# B&R Automation Studio project PLC code - cp (part 5)

#### MachineState.st
```iecst
ACTION MachineState:

	//Alignment photocells process
	tonAlignmentProcess.IN := (data.status.iSystemState=STP_CHECK_ALIGNMENT_STEP_3);
	tonAlignmentProcess.PT := t#2S;
	tonAlignmentProcess();

	CASE data.status.iSystemState OF

		STP_NOT_INITIALIZED:
			ResetCommands;
			ResetPhotocellAlignment;
			data.status.xReferencing :=	FALSE;

			IF NOT data.status.xReferenced THEN
				data.status.xSensorValidAlignPos := data.parameters.AlignmentProcess = STP_ALIGNMENT_NO_REQUIRED;
			END_IF

			RemoveOrderMoveAbsolute;
			SetStopOrder;
			IF xMotorStopped THEN
				RemoveStopOrder;
				CheckControllerReady;
				IF xControllerReady THEN
					data.status.iSystemState:=STP_POWER_ON;
				END_IF
			END_IF

		STP_POWER_ON:
			SetPowerOn;
			// It does HomeDirect to steppers when are power up is done
			CheckPowerOn;
			CASE data.parameters.MotorType OF
				STP_STEPPER:
					IF xPoweredOn AND NOT data.status.xReferenced THEN
						// Home Direct to enable movements
						data.status.iSystemState:=STP_HOME_DIR;

						// When Phocells are referenced and return from Zero (Man or Auto)
					ELSIF Stepper.Status.PowerOn AND StepperGear.Status.PowerOn AND data.status.xReferenced AND StepperGear.Status.PLCopenState.StandStill THEN
						data.status.iSystemState:=STP_GEARING;
					END_IF
				STP_ICLA:
					IF xPoweredOn THEN
						//Go directly to wait homing process
						data.status.iSystemState:=STP_GEARED;
					END_IF
			END_CASE

		STP_HOME_DIR:
			// Home position. Just send the order when the axis is ready
			IF Stepper.Status.PLCopenState.StandStill THEN
				Stepper.Parameter.HomePosition:=30;
				Stepper.Command.HomeDirect:=TRUE;
			END_IF
			IF StepperGear.Status.PLCopenState.StandStill THEN
				StepperGear.Parameter.HomePosition:=30;
				StepperGear.Command.HomeDirect:=TRUE;
			END_IF

			IF Stepper.Status.HomeOK AND StepperGear.Status.HomeOK THEN
				data.status.iSystemState:=STP_GEARING;
			END_IF

		STP_GEARING:
			StepperGear.Parameter.GearRatioNum:=1;
			StepperGear.Parameter.GearRationDen:=1;

			IF StepperGear.Status.PLCopenState.StandStill THEN
				StepperGear.Command.Move.GearIn:=TRUE;
			ELSIF StepperGear.Status.PLCopenState.SynchronizedMotion THEN
				data.status.iSystemState:=STP_GEARED;
			END_IF

		STP_GEARED:
			IF EDGEPOS(data.commandsSw.xReference) AND data.status.xAllPhotoInactive THEN
				data.commandsSw.xReference := FALSE;
				data.status.iSystemState := STP_HOMING_STEP_1;
			END_IF

			CheckMotorReady;
			IF data.status.xReferenced AND xMotorReady THEN
				CASE data.parameters.AlignmentProcess OF
					STP_ALIGNMENT_NO_REQUIRED:
						data.status.iSystemState := STP_STANDSTILL;

					STP_ALIGNMENT_REQUIRED:
						IF data.status.xSensorValidAlignPos THEN
							data.status.iSystemState := STP_STANDSTILL;
						ELSIF data.status.xReferencing THEN
							data.status.iSystemState := STP_SEARCH_ALIGNMENT_POS_STEP_1;
						END_IF
				END_CASE
			END_IF

			IF xMotorReady AND data.commands.Mode.xManual AND
				(data.ordersSw.xMoveDown OR data.ordersSw.xMoveUp) THEN
				data.status.iSystemState:=STP_JOGGING;
			END_IF

		STP_HOMING_STEP_1:
			data.status.xReferencing := TRUE;
			data.status.xReferenced	:= FALSE;

			IF data.parameters.xHomingEnabled THEN

				SetOrderGoingDown;

				//Stop going down when sensor to reference detects
				IF data.Inputs.Signals.xPhotoCells[data.parameters.iSensorToReference] THEN
					RemoveOrderGoingDown; // Launched stop movement

					//Once the jog is finished, we need to move up slowly to get the real position
					CheckMotorReady;
					IF xMotorReady THEN
						data.status.iSystemState := STP_HOMING_STEP_2;
					END_IF
				END_IF
			END_IF

		STP_HOMING_STEP_2:
			SetOrderGoingUp; // Launched movement

			//Moving slowly up to get the sensor again
			IF NOT data.Inputs.Signals.xPhotoCells[data.parameters.iSensorToReference] THEN
				// Movements finished
				RemoveOrderGoingUp; // Launched stop movement
				data.Alarms.xIncoherPhotocellSystem := FALSE;

				//Once the jog is finished, we need to gearOut to be able to do the Homing
				CheckMotorReady;
				IF xMotorReady THEN

					CASE data.parameters.MotorType OF
						STP_STEPPER:
							//Calculate the pulses of the HomingPosition
							MotorDriveUnit.HomePositionDesired:=data.parSw.rThicknessReference;
							MotorDriveUnit.Calculation:=CALC_HOMEPOS_PULSES;
							MotorDriveUnit();

							Stepper.Parameter.HomePosition := MotorDriveUnit.pulsesHomePositionDesired;
							StepperGear.Parameter.HomePosition := Stepper.Parameter.HomePosition;
							StepperGear.Command.Move.GearOut := TRUE;
							data.status.iSystemState := STP_HOMING_STEP_3;

						STP_ICLA:
							//Calculate the pulses of the HomingPosition
							MotorDriveUnit.HomePositionDesired:=(-1) * data.parSw.rThicknessReference;
							MotorDriveUnit.Calculation:=CALC_HOMEPOS_PULSES;
							MotorDriveUnit();

							IF Icla.Status.iActualVelocity = 0 THEN
								Icla.Parameter.Home.Position := REAL_TO_DINT(MotorDriveUnit.pulsesHomePositionDesired);
								Icla.Command.Home := TRUE;
							END_IF

							IF Icla.Status.xReferenced THEN data.status.iSystemState := STP_HOMING_STEP_3; END_IF

					END_CASE
				END_IF
			END_IF

		STP_HOMING_STEP_3:
			CASE data.parameters.MotorType OF
				STP_STEPPER:
					//Send a QuickStop to avoid the ContinuousMotion status after the GearOut
					StepperGear.Command.QuickStop := StepperGear.Status.PLCopenState.ContinuousMotion;

					IF Stepper.Status.PLCopenState.StandStill AND StepperGear.Status.PLCopenState.StandStill THEN
						// Home Direct
						Stepper.Command.HomeDirect:=TRUE;
						StepperGear.Command.HomeDirect:=TRUE;
						data.status.iSystemState := STP_HOMING_STEP_4;
					END_IF

				STP_ICLA:
					IF ABS(rPositionMotorMm - data.parSw.rThicknessReference) < 0.10 THEN
						//data.status.xReferencing := FALSE;
						data.status.xReferenced	:= TRUE;
						data.status.iSystemState := STP_GEARED;
					ELSE
						Icla.Command.Home := FALSE;
						data.status.iSystemState := STP_HOMING_STEP_2;
					END_IF
			END_CASE

		STP_HOMING_STEP_4:
			IF EDGEPOS(Stepper.Status.HomeOK AND StepperGear.Status.HomeOK) THEN
				data.status.xReferencing := FALSE;
				data.status.xReferenced	:= TRUE;
				data.status.iSystemState := STP_GEARING;
			END_IF

		STP_SEARCH_ALIGNMENT_POS_STEP_1:
			xAlignmentPositionSet := FALSE;
			SetOrderGoingUp;
			// Gauge is going to be higher than this position. Checking SensorToReference state from it.
			IF (rPositionMotorMm > data.parameters.rSensorPositionSearchAlignment) AND (data.Inputs.Signals.xPhotoCells[data.parameters.iSensorToReference]) THEN
				RemoveOrderGoingUp; // Launched stop movement
				data.status.iSystemState := STP_SEARCH_ALIGNMENT_POS_STEP_2;
			END_IF

		STP_SEARCH_ALIGNMENT_POS_STEP_2:
			SetOrderGoingUp; //Moving slowly up to get the sensor again
			IF NOT data.Inputs.Signals.xPhotoCells[data.parameters.iSensorToReference] THEN
				RemoveOrderGoingUp; // Launched stop movement
				rSensorPositionAlignmentMin := rPositionMotorMm;
				data.status.iSystemState := STP_SEARCH_ALIGNMENT_POS_STEP_3;
			END_IF

		STP_SEARCH_ALIGNMENT_POS_STEP_3:
			SetOrderGoingUp; //Moving slowly up to get the sensor again
			IF (data.Inputs.Signals.xPhotoCells[data.parameters.iSensorToReference]) THEN
				RemoveOrderGoingUp; // Launched stop movement
				rSensorPositionAlignmentMax := rPositionMotorMm;
				SetAlignmentPosition;
				data.status.rSensorPositionAlignment := rSensorPositionAlignment;
				data.status.xReferencing := FALSE;
				data.status.iSystemState := STP_STANDSTILL;
			END_IF

		STP_STANDSTILL:
			CheckAnyManualOrder;
			IF EDGEPOS(data.commandsSw.xReference) AND data.status.xAllPhotoInactive THEN
				data.commandsSw.xReference	:= FALSE;
				data.status.xReferenced	:= FALSE;
				data.status.xSensorValidAlignPos := FALSE;
				data.status.iSystemState	:= STP_HOMING_STEP_1;

			ELSIF data.commands.Mode.xManual AND xAnyManualOrder THEN
				data.status.iSystemState:=STP_JOGGING;

			ELSIF data.commands.Mode.xAuto THEN
				CASE data.parameters.AlignmentProcess OF
					STP_ALIGNMENT_NO_REQUIRED:
						data.status.iSystemState := STP_AUTO;

					STP_ALIGNMENT_REQUIRED:
						//First time machine goes to AUTO mode, to check alignment
						IF  data.status.xSensorValidAlignPos AND (NOT data.status.xAlignmentChecked) THEN
							data.status.iSystemState := STP_CHECK_ALIGNMENT_STEP_1;

						ELSIF data.status.xAlignmentChecked THEN
							data.status.iSystemState := STP_AUTO;
						END_IF
				END_CASE
			END_IF

		STP_JOGGING:
			// Stopping all
			IF tonMaxTimeJogging.Q THEN
				data.ordersSw.xMoveDown		:=	FALSE;
				data.ordersSw.xMoveUp		:=	FALSE;
			END_IF

			AssignJogOrders;

			CheckMotorReady;
			CheckAnyManualOrder;
			IF data.status.xReferenced AND xMotorReady AND NOT xAnyManualOrder THEN
				data.status.iSystemState	:= STP_STANDSTILL;

			ELSIF NOT data.status.xReferenced AND xMotorReady AND NOT xAnyManualOrder THEN
				data.status.iSystemState	:= STP_GEARED;

			END_IF

		STP_AUTO:
			IF NOT data.status.xInPosition THEN
				IF data.parameters.MotorType = STP_STEPPER THEN
					MotorDriveUnit.PositionDesired := rSensorPositionDesired;
				ELSE
					MotorDriveUnit.PositionDesired := (-1) * rSensorPositionDesired;
				END_IF
				MotorDriveUnit.Calculation := CALC_POS_PULSES;
				MotorDriveUnit();
				SetOrderMoveAbsolute;
				data.status.iSystemState := STP_RUNING;
			END_IF

		STP_CHECK_ALIGNMENT_STEP_1:
			//When the movement is finished
			IF data.parameters.MotorType = STP_STEPPER THEN
				MotorDriveUnit.PositionDesired := rSensorPositionAlignment;
			ELSE
				MotorDriveUnit.PositionDesired := (-1) * rSensorPositionAlignment;
			END_IF
			MotorDriveUnit.Calculation := CALC_POS_PULSES;
			MotorDriveUnit();
			SetOrderMoveAbsolute;
			data.status.iSystemState := STP_CHECK_ALIGNMENT_STEP_2;

		STP_CHECK_ALIGNMENT_STEP_2:
			//When the movement is finished
			IF (ABS(rPositionMotorMm-rSensorPositionAlignment)<0.25)  THEN
				data.status.iSystemState := STP_CHECK_ALIGNMENT_STEP_3;
			END_IF

			//Sensor alignment checking process cancelled when print order is set
			ReviewCancelCheckAlignment;

		STP_CHECK_ALIGNMENT_STEP_3:
			IF tonAlignmentProcess.Q THEN
				CheckPhotocellsAlignment;
				tonAlignmentProcess(IN := FALSE); //Clean the timer for next time in this stage

			//Due to issue DELOREAN-1129. Motor stays in this state. To exit, go to zero mode, then "xAlignmentChecked" is set to FALSE check process is executed when going to auto again.
			ELSIF data.status.xAlignmentChecked THEN
				data.status.iSystemState := STP_CHECK_ALIGNMENT_STEP_4;
			END_IF

			//Sensor alignment checking process cancelled when print order is set
			ReviewCancelCheckAlignment;

		STP_CHECK_ALIGNMENT_STEP_4:
			IF (NOT data.Alarms.xAlrCriticalPhotocellNotAligned) OR data.commands.Mode.xZero THEN
				data.status.iSystemState := STP_CHECK_ALIGNMENT_STEP_5;
			ELSIF data.commands.xErrorRst THEN
				ResetPhotocellAlignment;
				data.status.iSystemState := STP_CHECK_ALIGNMENT_STEP_3;
			END_IF

		STP_CHECK_ALIGNMENT_STEP_5:
			// Code from AUTO (previously from STP_CHECK_ALIGNMENT_STEP_4 to StandStill>>Auto
			IF NOT data.status.xInPosition THEN
				IF data.parameters.MotorType = STP_STEPPER THEN
					MotorDriveUnit.PositionDesired := rSensorPositionDesired;
				ELSE
					MotorDriveUnit.PositionDesired := (-1) * rSensorPositionDesired;
				END_IF
				MotorDriveUnit.Calculation := CALC_POS_PULSES;
				MotorDriveUnit();
				SetOrderMoveAbsolute;
				data.status.iSystemState := STP_CHECK_ALIGNMENT_STEP_6;
			END_IF

		STP_CHECK_ALIGNMENT_STEP_6:
			// Code from RUNNING. Previously from Auto>>Running
			//If the movement is finished or the desired position has changed
			tonMotorStopped(IN:=xMotorStopped, PT:=T#500ms);
			IF (data.status.xInPosition OR tonMotorStopped.Q) THEN
				RemoveOrderMoveAbsolute;
				data.status.iSystemState := STP_AUTO;
				tonMotorStopped(IN:=FALSE);
			END_IF

		STP_RUNING:
			//If the movement is finished or the desired position has changed
			tonMotorStopped(IN:=xMotorStopped, PT:=T#500ms);
			IF (data.status.xInPosition OR tonMotorStopped.Q) THEN
				RemoveOrderMoveAbsolute;
				data.status.iSystemState := STP_AUTO;
				tonMotorStopped(IN:=FALSE);
			END_IF

		STP_ERROR:
			ResetCommands;
			SetPowerOff;

			IF data.parameters.MotorType = STP_STEPPER THEN
				Stepper.Command.Reset := Stepper.Status.ControllerReady AND Stepper.Status.ErrorID<>0 AND data.commands.xErrorRst;
				Stepper.Command.ErrorAcknowledge :=	Stepper.Status.ErrorID<>0 AND data.commands.xErrorRst;

				StepperGear.Command.Reset := StepperGear.Status.ControllerReady AND StepperGear.Status.ErrorID<>0 AND data.commands.xErrorRst;
				StepperGear.Command.ErrorAcknowledge := StepperGear.Status.ErrorID<>0 AND data.commands.xErrorRst;
			END_IF

			data.status.xReferencing :=	FALSE;

			IF NOT data.status.xMotorError THEN data.status.iSystemState:=STP_NOT_INITIALIZED; END_IF;

	END_CASE

	//Sending nLaser to ERROR
	CASE data.parameters.MotorType OF
		STP_STEPPER:
			// Force state in Error/Zero state
			IF ((xAnyErrorStepper OR data.AlSummary.xAnyAlarm) AND (Stepper.Status.ErrorID<>31221)) OR tonTimeOutGearing.Q THEN
				data.status.iSystemState:=STP_ERROR;
			END_IF

		STP_ICLA:
			IF ((Icla.Status.iDriveStatus = ICLAST_ERROR) OR data.AlSummary.xAnyAlarm) THEN
				data.status.iSystemState:=STP_ERROR;
			END_IF
	END_CASE

	//In Zero mode it goes to not Init
	IF (data.commands.Mode.xZero) THEN
		data.status.iSystemState:=STP_NOT_INITIALIZED;
	END_IF;

	iReasonCheckingAlignment.0 := data.status.iSystemState = STP_CHECK_ALIGNMENT_STEP_1;
	iReasonCheckingAlignment.1 := data.status.iSystemState = STP_CHECK_ALIGNMENT_STEP_2;
	iReasonCheckingAlignment.2 := data.status.iSystemState = STP_CHECK_ALIGNMENT_STEP_3;
	iReasonCheckingAlignment.3 := data.status.iSystemState = STP_CHECK_ALIGNMENT_STEP_4;
	iReasonCheckingAlignment.4 := data.status.iSystemState = STP_CHECK_ALIGNMENT_STEP_5;
	iReasonCheckingAlignment.5 := data.status.iSystemState = STP_CHECK_ALIGNMENT_STEP_6;
	data.status.xCheckingAlignment := iReasonCheckingAlignment > 0;

	//Silvia: delay gearing motors.
	tonTimeOutGearing.IN:=data.status.iSystemState=STP_GEARING;
	tonTimeOutGearing.PT:=t#4s;
	tonTimeOutGearing();

	//Alarm excessive photecell activated
	tonMaxTimeJogging.IN:= (data.ordersSw.xMoveDown OR data.ordersSw.xMoveUp);
	tonMaxTimeJogging.PT:= T#5S;
	tonMaxTimeJogging();

	//Saving state history
	IF data.status.iSystemState<>StateHistory[0] THEN
		FOR iIndexHistory:=iHistoryLines TO 1 BY -1 DO
			StateHistory[iIndexHistory]:=StateHistory[iIndexHistory-1];
		END_FOR;
		StateHistory[0]:=data.status.iSystemState;
	END_IF

END_ACTION

ACTION ResetCommands:
	IF data.parameters.MotorType = STP_STEPPER THEN
		StepperGear.Command.Power      := FALSE;
		Stepper.Command.QuickStop	   := FALSE;
		StepperGear.Command.QuickStop  := FALSE;
		Stepper.Command.Jog.ContinuousPos	:=	FALSE;
		Stepper.Command.Jog.ContinuousNeg	:=	FALSE;
	ELSIF data.parameters.MotorType = STP_ICLA THEN
		Icla.Command.Enable := FALSE;
		Icla.Command.JogBackward := FALSE;
		Icla.Command.JogForward := FALSE;
		Icla.Command.MoveAbsolute := FALSE;
	END_IF
	data.commandsSw := ResetCommandsSw;
END_ACTION

ACTION CheckControllerReady:
	CASE data.parameters.MotorType OF
		STP_STEPPER:
			xControllerReady := Stepper.Status.ControllerReady AND StepperGear.Status.ControllerReady;
		STP_ICLA:
			xControllerReady := NOT Icla.Status.Error.Communication;
	END_CASE
END_ACTION

ACTION SetPowerOn:
	CASE data.parameters.MotorType OF
		STP_STEPPER:
			Stepper.Command.Power:=TRUE;
			StepperGear.Command.Power:=TRUE;
		STP_ICLA:
			Icla.Command.Enable := TRUE;
	END_CASE
END_ACTION

ACTION SetPowerOff:
	CASE data.parameters.MotorType OF
		STP_STEPPER:
			Stepper.Command.Power:=FALSE;
			StepperGear.Command.Power:=FALSE;
		STP_ICLA:
			Icla.Command.Enable := FALSE;
	END_CASE
END_ACTION

ACTION CheckPowerOn:
	CASE data.parameters.MotorType OF
		STP_STEPPER:
			xPoweredOn := Stepper.Status.PowerOn AND StepperGear.Status.PowerOn;
		STP_ICLA:
			xPoweredOn := Icla.Status.IclaStatus = AXISILE_POWER OR Icla.Status.IclaStatus = AXISILE_READY;
	END_CASE
END_ACTION

ACTION CheckMotorReady:
	CASE data.parameters.MotorType OF
		STP_STEPPER:
			xMotorReady := Stepper.Status.PLCopenState.StandStill AND StepperGear.Status.PLCopenState.SynchronizedMotion;
		STP_ICLA:
			xMotorReady := Icla.Status.iDriveStatus = ICLAST_ENABLE_OPERATION;
	END_CASE
END_ACTION

ACTION SetOrderGoingDown:
	CASE data.parameters.MotorType OF
		STP_STEPPER:
			Stepper.Command.Jog.ContinuousNeg := TRUE;

		STP_ICLA:
			Icla.Command.JogForward := TRUE;
	END_CASE
END_ACTION

ACTION RemoveOrderGoingDown:
	CASE data.parameters.MotorType OF
		STP_STEPPER:
			Stepper.Command.Jog.ContinuousNeg := FALSE;

		STP_ICLA:
			Icla.Command.JogForward := FALSE;
	END_CASE
END_ACTION

ACTION SetOrderGoingUp:
	CASE data.parameters.MotorType OF
		STP_STEPPER:
			Stepper.Command.Jog.ContinuousPos := TRUE;

		STP_ICLA:
			Icla.Command.JogBackward := TRUE;
	END_CASE
END_ACTION

ACTION RemoveOrderGoingUp:
	CASE data.parameters.MotorType OF
		STP_STEPPER:
			Stepper.Command.Jog.ContinuousPos := FALSE;

		STP_ICLA:
			Icla.Command.JogBackward := FALSE;
	END_CASE
END_ACTION

ACTION SetOrderMoveAbsolute:
	CASE data.parameters.MotorType OF
		STP_STEPPER:
			Stepper.Parameter.Position := MotorDriveUnit.pulsesPositionDesired;
			Stepper.Command.Move.Absolute := TRUE;

		STP_ICLA:
			Icla.Parameter.MoveAbsolute.Position := REAL_TO_DINT(MotorDriveUnit.pulsesPositionDesired);
			Icla.Command.MoveAbsolute := TRUE;
	END_CASE
END_ACTION

ACTION RemoveOrderMoveAbsolute:
	CASE data.parameters.MotorType OF
		STP_STEPPER:
			Stepper.Command.Move.Absolute := FALSE;

		STP_ICLA:
			Icla.Command.MoveAbsolute := FALSE;

	END_CASE
END_ACTION

ACTION SetStopOrder:
	CASE data.parameters.MotorType OF
		STP_STEPPER:
			Stepper.Command.QuickStop := TRUE;

		STP_ICLA:
			Icla.Command.Stop := TRUE;

	END_CASE
END_ACTION

ACTION RemoveStopOrder:
	CASE data.parameters.MotorType OF
		STP_STEPPER:
			Stepper.Command.QuickStop := FALSE;

		STP_ICLA:
			Icla.Command.Stop := FALSE;

	END_CASE
END_ACTION

ACTION AssignJogOrders:
	CASE data.parameters.MotorType OF
		STP_STEPPER:
			Stepper.Command.Jog.ContinuousPos	:=	data.ordersSw.xMoveUp;
			Stepper.Command.Jog.ContinuousNeg	:=	data.ordersSw.xMoveDown AND NOT Stepper.Command.Jog.ContinuousPos;

		STP_ICLA:
			Icla.Command.JogForward := data.ordersSw.xMoveDown AND NOT data.ordersSw.xMoveUp;
			Icla.Command.JogBackward := NOT data.ordersSw.xMoveDown AND data.ordersSw.xMoveUp;

	END_CASE
END_ACTION

ACTION CheckAnyManualOrder:
	xAnyManualOrder := data.ordersSw.xMoveUp OR data.ordersSw.xMoveDown;
END_ACTION

ACTION SetAlignmentPosition:
	rSensorPositionAlignment := (rSensorPositionAlignmentMax + rSensorPositionAlignmentMin)/2;
	data.status.xSensorValidAlignPos := (data.parameters.rSensorMechPositionAlignmentMin < rSensorPositionAlignment) AND (rSensorPositionAlignment < data.parameters.rSensorMechPositionAlignmentMax);
	xAlignmentPositionSet := rSensorPositionAlignment>0;
END_ACTION

ACTION CheckPhotocellsAlignment:
	FOR iIndexSensor:=1 TO data.parameters.iSensorQuantity DO
		data.status.xPhotoCellsNotAligned[iIndexSensor] := data.Inputs.Signals.xPhotoCells[iIndexSensor];
	END_FOR

	data.status.xAlignmentChecked := TRUE;
END_ACTION

ACTION ResetPhotocellAlignment:
	data.status.xAlignmentChecked := FALSE;
END_ACTION

ACTION CancelAlignment:
	data.status.xAlignmentChecked := TRUE;
END_ACTION

ACTION ReviewCancelCheckAlignment:
	IF (data.commands.xCancelAlignmentCheck) THEN
		CancelAlignment;
		RemoveOrderMoveAbsolute; //Allow a new edge and going to final position
		SetStopOrder;
		IF xMotorStopped THEN
			RemoveStopOrder;
			data.status.iSystemState:=STP_STANDSTILL;
		END_IF
	END_IF
END_ACTION
```

#### Motors.st
```iecst
ACTION DataToMotors:

	data.parSw.rMechOffset:=LIMIT(-1,data.parSw.rMechOffset, 1);

	IF data.parameters.MotorType = STP_STEPPER THEN
		StepperGear.Parameter.Direction	:= Stepper.Parameter.Direction; 	(* Step for a StepByStep movement *) (*Take carewith relative movements!!!!*)
	END_IF

	rJogSpeedSetPoint:=data.parameters.JogSpeed;

	//Drive Unit Data Managment
	MotorDriveUnit.TransmissionData := data.parameters.DriveUnit;

	MotorDriveUnit.SpeedDesired:=data.parameters.Speed;
	MotorDriveUnit.Calculation:=CALC_SPEED_PULSES;
	MotorDriveUnit();

	MotorDriveUnit.JogSpeedDesired:=rJogSpeedSetPoint;
	MotorDriveUnit.Calculation:=CALC_JOGSPEED_PULSES;
	MotorDriveUnit();

	MotorDriveUnit.AccelerationDesired:=data.parameters.Acceleration;
	MotorDriveUnit.Calculation:=CALC_ACC_PULSES;
	MotorDriveUnit();

	AssignDataToMotors;

END_ACTION

ACTION AssignDataToMotors:

	CASE data.parameters.MotorType OF
		STP_STEPPER:

			//Speed
			Stepper.Parameter.Speed:=MotorDriveUnit.pulsesSpeedDesired;
			StepperGear.Parameter.Speed := Stepper.Parameter.Speed;

			//Jog Speed
			Stepper.Parameter.JogSpeed:=MotorDriveUnit.pulsesJogSpeedDesired;
			StepperGear.Parameter.JogSpeed:=Stepper.Parameter.JogSpeed;

			//Acceleration
			Stepper.Parameter.Acceleration := MotorDriveUnit.pulsesAccelerationDesired;
			Stepper.Parameter.Deceleration := Stepper.Parameter.Acceleration;
			StepperGear.Parameter.Acceleration := Stepper.Parameter.Acceleration;
			StepperGear.Parameter.Deceleration := Stepper.Parameter.Deceleration;

			//Reset
			Stepper.Command.ErrorAcknowledge:= Stepper.Status.ErrorID=31221 OR (Stepper.Status.ErrorID = 29207) OR (Stepper.Status.ErrorID = 29205); // Disturbance in cables?
			StepperGear.Command.ErrorAcknowledge:= StepperGear.Status.ErrorID=31221 OR (Stepper.Status.ErrorID = 29207) OR (Stepper.Status.ErrorID = 29205);

			//Enable Permanent Encoder Data
			Stepper.Parameter.Init.xEnabledPermEncData:=TRUE;
			StepperGear.Parameter.Init.xEnabledPermEncData:=TRUE;

		STP_ICLA:

			//Enable
			Icla.Command.Enable:= Icla.Status.iDriveStatus <> ICLAST_ERROR;

			//Speed
			Icla.Parameter.MoveAbsolute.Velocity := REAL_TO_UINT(MotorDriveUnit.pulsesSpeedDesired);

			//Jog Speed
			Icla.Parameter.Jog.VeloSlow := REAL_TO_UINT(MotorDriveUnit.pulsesJogSpeedDesired);
			Icla.Command.JogFastSpeed := FALSE;

			//Acceleration
			Icla.Parameter.iAcceleration := REAL_TO_UINT(MotorDriveUnit.pulsesAccelerationDesired);

			//Reset
			Icla.Command.Reset := 	data.commands.xResetMotor OR 	(data.commands.xErrorRst AND
																	Icla.Status.IclaStatus <> AXISILE_MOVE_ABSOLUTE AND
																	Icla.Status.IclaStatus <> AXISILE_JOG AND
																	Icla.Status.IclaStatus <> AXISILE_HOMING);

			data.status.Icla.xIsMoving := Icla.Status.iActualVelocity<>0;

	END_CASE

END_ACTION

ACTION DataFromMotors:

	CASE data.parameters.MotorType OF
		STP_STEPPER:
			// All manual movements are done with Jog, Photocells.status.xReferencing is done by Jog, could be it done by trigger?
			xAnyManualMovement:= Stepper.Status.PLCopenState.ContinuousMotion OR StepperGear.Status.PLCopenState.ContinuousMotion;

			MotorDriveUnit.pulsesDevice:=Stepper.Status.ActPosition;

			//Conversions
			MotorDriveUnit.Calculation:= CALC_POS_MM;
			MotorDriveUnit();
			rPositionMotorMm := MotorDriveUnit.PositionDevice;

			data.status.rPositionMotor := rPositionMotorMm;

			// Errrors assumed ?
			xAnyErrorStepper:=	(Stepper.Status.ErrorID<>0) OR (StepperGear.Status.ErrorID<>0);
			data.status.xMotorError:= xAnyErrorStepper AND (((Stepper.Status.ErrorID<>31221)AND (Stepper.Status.ErrorID<>29207) AND (Stepper.Status.ErrorID<>29205)) OR // It avoids data.status.xZero
															((StepperGear.Status.ErrorID<>31221)AND (StepperGear.Status.ErrorID<>29207) AND (StepperGear.Status.ErrorID<>29205)));
			data.status.iErrorId:=Stepper.Status.ErrorID;
			xMotorStopped := Stepper.Status.ActVelocity = 0;

			IF (Stepper.Status.ErrorID = 29205) OR (StepperGear.Status.ErrorID = 29205) THEN
				data.status.xReferenced := FALSE;
			END_IF

		STP_ICLA:
			xAnyManualMovement:= (Icla.Status.IclaStatus = AXISILE_JOG);

			MotorDriveUnit.pulsesDevice := DINT_TO_REAL(Icla.Status.iActualPosition);
			MotorDriveUnit.PulsesSpeedDevice:=Icla.Status.iActualVelocity;

			// Conversions
			MotorDriveUnit.Calculation:= CALC_POS_MM;
			MotorDriveUnit();
			rPositionMotorMm := (-1)*MotorDriveUnit.PositionDevice;

			data.status.rPositionMotor := rPositionMotorMm;

			// Errors
			data.status.xMotorError:= Icla.Status.Error.Communication OR Icla.Status.Error.ErrorNumber<>0; // It avoids data.status.xZero
			data.status.Icla.iErrorId:= Icla.Status.Error.ErrorNumber;

			data.status.Icla.rCurrentPosition:= Icla.Status.iActualPosition;
			data.status.Icla.rCurrentVel:= Icla.Status.iActualVelocity;

			xMotorStopped := Icla.Status.iActualVelocity = 0;

	END_CASE

	//Sending upwards the information of the location of the sensors
	data.status.xInPosition := ABS(rPositionMotorMm - rSensorPositionDesired) < 0.10;
	data.status.xAboveSetPoint := rPositionMotorMm >= rSensorPositionDesired + 0.10;
	data.status.xBelowSetPoint := rPositionMotorMm <= rSensorPositionDesired - 0.10;

	//To avoid change rBarsPosition value while motor is being positioned to new position setpoint. Issue discovered while changing thickness from 2 to 10mm at 90m/min
	//Bars were going down executing little steps because "rMaxPosition" was written every scan cycle with a new value coming due to this "rPositionWithOffset"
	IF data.status.xInPosition THEN
		data.status.rPositionWithOffset := rPositionMotorMm - data.parSw.rMechOffset;
	END_IF

	MotorDriveUnit.Calculation:= CALC_SPEED_MM;
	MotorDriveUnit();

END_ACTION
```

### Program Logical/ExtPack/_Media/nSensorCtrl/nSensorCtrl_v2/nSensorCtrl_Fast (IEC)

#### nSensorCtrl_Fast.st - Init, cyclic, exit code
```iecst
PROGRAM _CYCLIC

	//Main data assignation
	data 	ACCESS ADR (gPhotoCells);

	//Not execute the code if the nSensor system is not installed
	IF NOT data.status.xInstalled THEN	RETURN;	END_IF

	//If in not Simulation check the pointers and assign data
	IF gMachine.St.HwData.Family <> FAMILY_BRAUTOMATIONRUNTIME THEN

		// Check value for all sensors considered
		FOR iIndexCheckSensor := 1 TO data.parameters.iSensorQuantity DO
			IF (data.Inputs.Signals.pInput[iIndexCheckSensor] <> 0) THEN
				pointerValue ACCESS (data.Inputs.Signals.pInput[iIndexCheckSensor]);
				data.Inputs.Signals.xPhotoCells[iIndexCheckSensor] := NOT pointerValue;
			ELSE
				RETURN;
			END_IF
		END_FOR

	END_IF

	xRecordMaxPosition := data.commands.xRecordMaxPosition;
	IF xRecordMaxPosition THEN
		rMaxPosition := MAX(data.parameters.rMediaThickness, data.status.rPositionWithOffset);
		rBarPosition := rMaxPosition;
	END_IF

	IF data.status.xSensorsPositionedRelativeToBar THEN
		iFirstSensorToCheck:=data.status.iSensorToApplyOffset;
	ELSE
		iFirstSensorToCheck:=data.parameters.iSensorToReference;
	END_IF

	xMountedMediaDetected := FALSE;
	xMediaToRejectDetected := FALSE;

	// Checking Mounted data if machine is in conditions to Check
	IF data.commands.xCheckMounted THEN
		//Just above the Sensor for reference. Sensors below not used. Just to know if media inside (parameters.iSensorToReference)
		//Running photocells from the one assemblied closest to printer's entry and highest located. In case mountedTile alarm, will be active at first iterations
		FOR iIndexSensor:=iFirstSensorToCheck TO data.parameters.iSensorQuantity DO
			IF data.Inputs.Signals.xPhotoCells[iIndexSensor] THEN
				//Define the position of the bars
				IF iIndexSensor<>data.parameters.iSensorQuantity THEN
					IF data.status.xSensorsPositionedRelativeToBar THEN
						rBarPosition := data.status.rOffsetToApplyToBarsPosition + data.parameters.rOffsetRelToBar + data.parameters.Sensors[iIndexSensor+1].rDistanceRelativeToFirstSensor + data.parameters.Sensors[iIndexSensor+1].rSafetyOffset;
					ELSE
						rBarPosition := data.parameters.rMediaThickness + data.parameters.Sensors[iIndexSensor+1].rDistanceRelativeToFirstSensor + data.parameters.rOffsetPosition + data.parameters.Sensors[iIndexSensor+1].rSafetyOffset;
					END_IF
				END_IF

				// Define the States to raise Mounted Alarms
				iStatusCheckMounted.0 := data.status.iSystemState = STP_AUTO;
				iStatusCheckMounted.1 := data.status.iSystemState = STP_RUNING;

				IF iStatusCheckMounted > 0 THEN
					//Raise the Mounted alarm if sensor active and it is configured to raise mounted.
					IF data.parameters.xRaiseMountedJustBelowPrePrint THEN
						// This is the case for Cube_Alpha, where was important add more safety to do not raise the alarm in the wrong position and with nonsense
						IF data.parameters.Sensors[iIndexSensor].xMountedMedia AND data.status.rPositionMotor < data.parameters.rPrePrintPosition + 0.5 THEN
							// This alarm has to be raised here to avoid resetting it and move out the mounted media
							IF NOT data.commands.xMountedMediaInside THEN
								data.Alarms.xMountedTile:= TRUE;
							END_IF
							xMountedMediaDetected := TRUE;
							EXIT;
						END_IF
					ELSE
						// Previous behavior not tacking into account Cube machines
						IF data.parameters.Sensors[iIndexSensor].xMountedMedia THEN
							// This alarm has to be raised here to avoid resetting it and move out the mounted media
							IF NOT data.commands.xMountedMediaInside THEN
								data.Alarms.xMountedTile:= TRUE;
							END_IF
							xMountedMediaDetected := TRUE;
							EXIT;
						END_IF
					END_IF
				END_IF

				//Marking media to be rejected when any laser configured to do that. Due to low quality printing when bars moving up upper of sensor's height
				IF data.parSw.Sensors[iIndexSensor].xToRejectMedia THEN
					xMediaToRejectDetected := TRUE;
				END_IF

			END_IF

		END_FOR

	ELSE
		//data.status.xMediaToRejectDetected := FALSE;
	END_IF

	// Data has to be treated in the slow program to be sure to read the information in all fast programs
	IF xMountedMediaDetected (*AND NOT data._Internal.xMountedMediaTreated*) THEN
		data.status.xMountedMediaDetected := TRUE;
	ELSIF NOT xMountedMediaDetected AND data._Internal.xMountedMediaTreated THEN
		data.status.xMountedMediaDetected := FALSE;
	END_IF

	// Data has to be treated in the slow program to be sure to read the information in all fast programs
	IF xMediaToRejectDetected (*AND NOT data._Internal.xMediaToRejectTreated*) THEN
		data.status.xMediaToRejectDetected := TRUE;
	ELSIF NOT xMediaToRejectDetected AND data._Internal.xMediaToRejectTreated THEN
		data.status.xMediaToRejectDetected := FALSE;
	END_IF

	data.status.rBarsPosition := rBarPosition;
	data.status.xLowPieceDetect := data.Inputs.Signals.xPhotoCells[1];

	// If the bars are in high position, do not register photocelles activation/deactivation
	IF data.status.rPositionMotor > (data.parameters.rPrePrintPosition + 0.5) THEN
		RETURN;
	END_IF

	IF EDGEPOS(data.Inputs.Signals.xPhotoCells[2]) THEN LogRaiseSensor2; END_IF
	IF EDGEPOS(data.Inputs.Signals.xPhotoCells[3]) THEN LogRaiseSensor3; END_IF
	IF EDGEPOS(data.Inputs.Signals.xPhotoCells[4]) THEN LogRaiseSensor4; END_IF
	IF EDGEPOS(data.Inputs.Signals.xPhotoCells[5]) THEN LogRaiseSensor5; END_IF
	IF EDGEPOS(data.Inputs.Signals.xPhotoCells[6]) THEN LogRaiseSensor6; END_IF

	IF EDGENEG(data.Inputs.Signals.xPhotoCells[2]) THEN LogLowerSensor2; END_IF
	IF EDGENEG(data.Inputs.Signals.xPhotoCells[3]) THEN LogLowerSensor3; END_IF
	IF EDGENEG(data.Inputs.Signals.xPhotoCells[4]) THEN LogLowerSensor4; END_IF
	IF EDGENEG(data.Inputs.Signals.xPhotoCells[5]) THEN LogLowerSensor5; END_IF
	IF EDGENEG(data.Inputs.Signals.xPhotoCells[6]) THEN LogLowerSensor6; END_IF

END_PROGRAM
```

#### EventLog.st
```iecst
ACTION LogRaiseSensor2:

	stRaiseSensor2.Source := ELOG_TYPE_DETECTION;
	stRaiseSensor2.Severity:= ELOG_SEVERITY_INFO;
	stRaiseSensor2.Facility:= 2;
	stRaiseSensor2.ErrorCode:=0;

	stRaiseSensor2.Text := 'nSensor. Raised Sensor2';

	gEventLogLoader(EventData := ADR(stRaiseSensor2));

END_ACTION

ACTION LogLowerSensor2:

	stLowerSensor2.Source := ELOG_TYPE_DETECTION;
	stLowerSensor2.Severity:= ELOG_SEVERITY_INFO;
	stLowerSensor2.Facility:= 2;
	stLowerSensor2.ErrorCode:=0;

	stLowerSensor2.Text := 'nSensor. Lowered Sensor2';

	gEventLogLoader(EventData := ADR(stLowerSensor2));

END_ACTION

ACTION LogRaiseSensor3:

	stRaiseSensor3.Source := ELOG_TYPE_DETECTION;
	stRaiseSensor3.Severity:= ELOG_SEVERITY_INFO;
	stRaiseSensor3.Facility:= 3;
	stRaiseSensor3.ErrorCode:=0;

	stRaiseSensor3.Text := 'nSensor. Raised Sensor3';

	gEventLogLoader(EventData := ADR(stRaiseSensor3));

END_ACTION

ACTION LogLowerSensor3:

	stLowerSensor3.Source := ELOG_TYPE_DETECTION;
	stLowerSensor3.Severity:= ELOG_SEVERITY_INFO;
	stLowerSensor3.Facility:= 3;
	stLowerSensor3.ErrorCode:=0;

	stLowerSensor3.Text := 'nSensor. Lowered Sensor3';

	gEventLogLoader(EventData := ADR(stLowerSensor3));

END_ACTION

ACTION LogRaiseSensor4:

	stRaiseSensor4.Source := ELOG_TYPE_DETECTION;
	stRaiseSensor4.Severity:= ELOG_SEVERITY_INFO;
	stRaiseSensor4.Facility:= 4;
	stRaiseSensor4.ErrorCode:=0;

	stRaiseSensor4.Text := 'nSensor. Raised Sensor4';

	gEventLogLoader(EventData := ADR(stRaiseSensor4));

END_ACTION

ACTION LogLowerSensor4:

	stLowerSensor4.Source := ELOG_TYPE_DETECTION;
	stLowerSensor4.Severity:= ELOG_SEVERITY_INFO;
	stLowerSensor4.Facility:= 4;
	stLowerSensor4.ErrorCode:=0;

	stLowerSensor4.Text := 'nSensor. Lowered Sensor4';

	gEventLogLoader(EventData := ADR(stLowerSensor4));

END_ACTION

ACTION LogRaiseSensor5:

	stRaiseSensor5.Source := ELOG_TYPE_DETECTION;
	stRaiseSensor5.Severity:= ELOG_SEVERITY_INFO;
	stRaiseSensor5.Facility:= 5;
	stRaiseSensor5.ErrorCode:=0;

	stRaiseSensor5.Text := 'nSensor. Raised Sensor5';

	gEventLogLoader(EventData := ADR(stRaiseSensor5));

END_ACTION

ACTION LogLowerSensor5:

	stLowerSensor5.Source := ELOG_TYPE_DETECTION;
	stLowerSensor5.Severity:= ELOG_SEVERITY_INFO;
	stLowerSensor5.Facility:= 5;
	stLowerSensor5.ErrorCode:=0;

	stLowerSensor5.Text := 'nSensor. Lowered Sensor5';

	gEventLogLoader(EventData := ADR(stLowerSensor5));

END_ACTION

ACTION LogRaiseSensor6:

	stRaiseSensor6.Source := ELOG_TYPE_DETECTION;
	stRaiseSensor6.Severity:= ELOG_SEVERITY_INFO;
	stRaiseSensor6.Facility:= 6;
	stRaiseSensor6.ErrorCode:=0;

	stRaiseSensor6.Text := 'nSensor. Raised Sensor6';

	gEventLogLoader(EventData := ADR(stRaiseSensor6));

END_ACTION

ACTION LogLowerSensor6:

	stLowerSensor6.Source := ELOG_TYPE_DETECTION;
	stLowerSensor6.Severity:= ELOG_SEVERITY_INFO;
	stLowerSensor6.Facility:= 6;
	stLowerSensor6.ErrorCode:=0;

	stLowerSensor6.Text := 'nSensor. Lowered Sensor6';

	gEventLogLoader(EventData := ADR(stLowerSensor6));

END_ACTION
```

#### nSensorCtrl_Fast.var - Local variables
```iecst
VAR
	data : REFERENCE TO nSensors_typ;
	rMaxPosition : REAL;
	rBarPosition : REAL;
	iFirstSensorToCheck : USINT;
	iIndexSensor : USINT;
	xRecordMaxPosition : BOOL; (*Variable to allow to record the max position*)
	iStatusCheckMounted : UINT;
	xMountedMediaDetected : BOOL;
	xMediaToRejectDetected : BOOL;
	iIndexCheckSensor : USINT;
	pointerValue : REFERENCE TO BOOL;
	stRaiseSensor1 : EventLog_typ;
	stLowerSensor1 : EventLog_typ;
	stRaiseSensor2 : EventLog_typ;
	stLowerSensor2 : EventLog_typ;
	stRaiseSensor3 : EventLog_typ;
	stLowerSensor3 : EventLog_typ;
	stRaiseSensor4 : EventLog_typ;
	stLowerSensor4 : EventLog_typ;
	stRaiseSensor5 : EventLog_typ;
	stLowerSensor5 : EventLog_typ;
	stRaiseSensor6 : EventLog_typ;
	stLowerSensor6 : EventLog_typ;
	stRaiseSensor7 : EventLog_typ;
	stLowerSensor7 : EventLog_typ;

END_VAR
```

### Program Logical/ExtPack/_Media/nSensorCtrl/nSensorSim/nSensorSim_v1/nSensorSim (IEC)

#### nSensorSim.var - Local variables
```iecst
VAR
	data : REFERENCE TO nSensors_typ;
	iIndexSensor : USINT;
	rGaugeHeightTillHole : REAL;
	tonHomingDown : TON;
	tonHomingUp : TON;
END_VAR
```

### Library Logical/ExtPack/_Media/ThicknessCtrl/ThickLib (IEC)

#### ThickLib.typ - local structure
```iecst
TYPE
	stThicknessCtrl_MediaPosStatus : 	STRUCT
		Media : stThicknessCtrl_MediaConfig;
		HeadPosition : UDINT; (*Position of the head of the media in cm*)
		TailPosition : UDINT; (*Position of the tail of the media in cm*)
		iIndexMediaEnergy : USINT; (*Index of the MediaEnergy information in the fixed cells*)
		pMediaEnery : UDINT; (*Pointer to the MediaEnergy information. It is in fixed cells in an array*)
	END_STRUCT;
	stThickCtrl_EnergyMedia : 	STRUCT  (*THIS STRUCTURE IS USED IN OPCUA METHODS. MODIFY IT NEEDS TO UPDATE SOFTWARE CODE!!!!!!    >>>Data coming directly from Energy Communications*)
		MediaData : stThicknessCtrl_MediaConfig;
		Energy : stThickCtrl_Energy;
	END_STRUCT;
	stThickCtrl_Energy : 	STRUCT  (*/// Data coming directly from Energy Communications*)
		iPower : ARRAY[0..THICKENERGY_MAX_PROCESS_ITEMS,0..THICKENERGY_MAX_CROSS_ITEMS]OF USINT; (*The Energy needs the media to be cured. Led or Dry*)
	END_STRUCT;
	stThicknessCtrl_MediaConfig : 	STRUCT  (*THIS STRUCTURE IS USED IN OPCUA METHODS. MODIFY IT NEEDS TO UPDATE SOFTWARE CODE!!!!!!*)
		id : DINT; (*Identificator of the board*)
		iLine : USINT; (*Line where the media will arrive to the printer [1, 2, ..]*)
		xHasClear : BOOL; (*The media document has opv ink*)
		xHasWhite : BOOL; (*The media document has white color*)
		rThickness : REAL; (*Media thickness to print from gui in mm*)
		rMargin : REAL; (*Printing Margin from the real media thickness in mm*)
		rWidth : REAL; (*Media width in mm. Cross direction*)
		rLength : REAL; (*Media length in mm. Process direction*)
		rCrossOffset : REAL; (*Document offset position in mm. From the center of the belt*)
		rDocWidth : REAL; (*Document width in mm. Cross direction*)
		rDocLength : REAL; (*Document length in mm. Process direction*)
		rDocCrossOffset : REAL; (*Document offset position in mm. From the center of the belt*)
		rDocProcessOffset : REAL; (*Document offset position in mm from head of substrate. From the head of the substrate. Positive through inside the substrate*)
	END_STRUCT;
	stThickCtrl_TrackingEventType :
		(
		HEAD_UNDEFINED,
		HEAD_DETECTED,
		TAIL_DETECTED,
		START_REJECTING_ALL,
		END_REJECTING_ALL,
		START_HOLDREJEC,
		END_HOLDREJECT
		);
	stThicknessCtrl_TrackingEvent : 	STRUCT  (*For now just a copy of ALL parameters*)
		diBeltPosition : UDINT := 0; (*Value of the belt position when detecting the event*)
		diDistanceToPrevious : UDINT := 0; (*Value of the belt position difference with the previous one. Wrong values with events not in cero (as HoldReject)*)
		Event : stThickCtrl_TrackingEventType := HEAD_UNDEFINED;
	END_STRUCT;
	ThicknessMountedDetectionType :
		(
		THICKMOUNT_UNDEFINED,
		THICKMOUNT_THICKNESS_RELATIVE,
		THICKMOUNT_ABSOLUTE
		);
END_TYPE
```

#### ThickLib.fun - Exported functions and function blocks
```iecst
{REDUND_ERROR} FUNCTION LoadMediaFromFastDataLine : BOOL (*Loading Fast data in an array to an array of tracking data. Using USINT array to load differente lines*) (*$GROUP=User,$CAT=User,$GROUPICON=User.png,$CATICON=User.png*)
	VAR_INPUT
		newValues : REFERENCE TO ARRAY[0..THICK_MAX_UPDATE_VALUES] OF BOOL; (*Array of the new Fast values*)
		fastValues : REAL; (*Total fast values loaded in the fast array*)
		indexLine : USINT; (*Number of the bit where to store the data in the tracking array*)
		positionsToRunArray : UINT; (*The positions to run the array. Corresponds the position to load data from fast in slow. Depending on the speed of the belt*)
		sensorPosition : UINT; (*Position of the sensor to insert the new data properly*)
		valuesTracking : REFERENCE TO ARRAY[0..iMAXTRACKINGARRAY] OF USINT; (*values tracked. 1cm per position*)
	END_VAR
	VAR
		iIndexArray : UINT;
		iIndexNewMediaArray : UINT;
		bitLine : USINT;
		rValuesPerPosition : REAL;
		iFirstIndex : UINT;
		iLastIndex : UINT;
	END_VAR
END_FUNCTION

{REDUND_ERROR} FUNCTION LoadMediaFromFastDataBool : BOOL (*Loading Fast data in an array to an array of tracking data. Using BOOL array to load individual data*) (*$GROUP=User,$CAT=User,$GROUPICON=User.png,$CATICON=User.png*)
	VAR_INPUT
		newValues : REFERENCE TO ARRAY[0..THICK_MAX_UPDATE_VALUES] OF BOOL; (*Array of the new Fast values*)
		fastValues : REAL; (*Total fast values loaded in the fast array*)
		positionsToRunArray : UINT; (*The positions to run the array. Corresponds the position to load data from fast in slow. Depending on the speed of the belt*)
		sensorPosition : UINT; (*Position of the sensor to insert the new data properly*)
		valuesTracking : REFERENCE TO ARRAY[0..iMAXTRACKINGARRAY] OF BOOL; (*values tracked. 1cm per position*)
	END_VAR
	VAR
		iIndexArray : UINT;
		iIndexNewMediaArray : UINT;
		rValuesPerPosition : REAL;
		iFirstIndex : UINT;
		iLastIndex : UINT;
	END_VAR
END_FUNCTION

{REDUND_ERROR} FUNCTION CheckFilteredMediaLine : BOOL (*Review if the values in a trackignArray is consistent. Using USINT array to load differente lines*) (*$GROUP=User,$CAT=User,$GROUPICON=User.png,$CATICON=User.png*)
	VAR_INPUT
		valuesTracking : REFERENCE TO ARRAY[0..iMAXTRACKINGARRAY] OF USINT; (*values tracked. 1cm per position*)
		indexLine : USINT; (*Number of the bit where to store the data in the tracking array*)
		sensorPosition : UINT; (*Position of the sensor to insert the new data properly*)
		mediaFilter : UINT; (*Filter to consider data consistent*)
	END_VAR
	VAR
		iIndexArray : UINT;
		bitLine : USINT;
		xFilteredData : BOOL;
	END_VAR
END_FUNCTION

{REDUND_ERROR} FUNCTION CheckFilteredMediaBool : BOOL (*Review if the values in a trackignArray is consistent. Using BOOL array to load individual data*) (*$GROUP=User,$CAT=User,$GROUPICON=User.png,$CATICON=User.png*)
	VAR_INPUT
		valuesTracking : REFERENCE TO ARRAY[0..iMAXTRACKINGARRAY] OF BOOL; (*values tracked. 1cm per position*)
		sensorPosition : UINT; (*Position of the sensor to insert the new data properly*)
		mediaFilter : UINT; (*Filter to consider data consistent*)
	END_VAR
	VAR
		iIndexArray : UINT;
		xFilteredData : BOOL;
	END_VAR
END_FUNCTION

FUNCTION ReviewMediaTrackingInPosition : BOOL (*Review if any element in the array is inside de window*)
	VAR_INPUT
		ArrayOfMedia : REFERENCE TO ARRAY[0..THICK_MEDIATRACKING_MAX_MEDIA] OF stThicknessCtrl_MediaPosStatus;
		TotalElementsInside : UINT; (*Total elements inside the array*)
		iStartWindow : UINT;
		iEndWindow : UINT;
		xIsWhite : BOOL;
	END_VAR
	VAR
		iIndexArray : UINT;
		xMediaInPosition : BOOL;
	END_VAR
END_FUNCTION

FUNCTION RevMediaTrackingEnergyInPos : BOOL (*Review if any element in the array is inside de window and calculate the Energy needed*)
	VAR_INPUT
		ArrayOfMedia : REFERENCE TO ARRAY[0..THICK_MEDIATRACKING_MAX_MEDIA] OF stThicknessCtrl_MediaPosStatus;
		TotalElementsInside : UINT; (*Total elements inside the array*)
		iStartWindow : INT; (*Distance in cm*)
		iEndWindow : INT; (*Distance in cm*)
		iTotalLamps : USINT;
		rLampWidth : REAL; (*Width of each lamp. Value in mm*)
		rLampOffset : REAL; (*Offset of the first lamp considering the center of the belt as 0. Positive to operator side. Value in mm*)
		rLampOverlap : REAL; (*Overlap to consider as extra width for each lamp. Value in mm*)
		iMinIntensity : INT; (*Minimum Intensity*)
	END_VAR
	VAR_IN_OUT
		iIntensity : ARRAY[0..THICKENERGY_MAX_LAMPS] OF INT; (*Data starting in index 1*)
	END_VAR
	VAR
		iIndexArray : UINT;
		Intensity : ARRAY[0..THICKENERGY_MAX_LAMPS] OF INT; (*Data starting in index 0*)
		diPosStartMedia : DINT;
		diPosEndMedia : DINT;
	END_VAR
END_FUNCTION

FUNCTION RevMediaTrackingEnergyInPosItem : BOOL (*Review if any element in the array is inside de window and calculate the Energy needed*)
	VAR_INPUT
		MediaData : REFERENCE TO stThicknessCtrl_MediaPosStatus;
		EnergyData : REFERENCE TO stThickCtrl_Energy;
		iStartWindow : INT; (*Distance in cm*)
		iEndWindow : INT; (*Distance in cm*)
		rLampWidth : REAL; (*Width of each lamp. Value in mm*)
		rLampOffset : REAL; (*Offset of the first lamp considering the center of the belt as 0. Positive to operator side. Value in mm*)
		rLampOverlap : REAL; (*Overlap to consider as extra width for each lamp. Value in mm*)
	END_VAR
	VAR_IN_OUT
		iIntensity : ARRAY[0..THICKENERGY_MAX_LAMPS] OF INT;
	END_VAR
	VAR
		iIndexCross : UINT;
		iIndexProcess : UINT;
		iIndexLamp : UINT;
		iFirstLamp : UINT; (*Starting with 0. The first lamp is index 0*)
		iLastLamp : UINT;
		rOffsetStartDocument : REAL; (*Position in mm to the center of the belt*)
		Intensity : ARRAY[0..THICKENERGY_MAX_LAMPS] OF INT;
		iLampIntensity : INT;
		iFirstCrossSection : INT;
		iLastCrossSection : INT;
		iFirstProcessSection : INT;
		iLastProcessSection : INT;
	END_VAR
END_FUNCTION

{REDUND_ERROR} FUNCTION AddMediaTrackingEvents : BOOL (*Loading Fast data in an array to an array of tracking data. Using USINT array to load differente lines*) (*$GROUP=User,$CAT=User,$GROUPICON=User.png,$CATICON=User.png*)
	VAR_INPUT
		diBeltPosition : UDINT; (*Total Position of the belt when occurring the event*)
		EventType : stThickCtrl_TrackingEventType; (*Event Type*)
		pEventsTrackingArray : UDINT; (*Address of the array. Calling as ADR(myArray)*)
	END_VAR
	VAR
		iIndexArray : UINT;
		iIndexNewMediaArray : UINT;
		rValuesPerPosition : REAL;
		fakeElement : stThicknessCtrl_TrackingEvent;
		EventsArray : REFERENCE TO ARRAY[0..THICK_MAX_TRACKING_EVENTS] OF stThicknessCtrl_TrackingEvent;
	END_VAR
END_FUNCTION

FUNCTION CheckMediaToStack : UDINT (*Check if the Media sent to the stack is correct. If returning 0 everything is OK, if not returning the error code*)
	VAR_INPUT
		NewMedia : stThicknessCtrl_MediaConfig;
		xStackEnabled : BOOL;
		xDtpEnabled : BOOL;
		rMaxThickness : REAL;
		rMinWidth : REAL;
		rMaxWidth : REAL;
		rMinLength : REAL;
		rMaxLength : REAL;
		xStackLine1Full : BOOL;
		xStackLine2Full : BOOL;
	END_VAR
END_FUNCTION

FUNCTION CheckLineToStack : UDINT (*Check if the Line to stack is correct. If returning 0 everything is OK, if not returning the error code*)
	VAR_INPUT
		iLine : USINT;
		xStackEnabled : BOOL;
		xDtpEnabled : BOOL;
	END_VAR
END_FUNCTION

FUNCTION CheckEnabledStack : UDINT (*Check if the Line to stack is correct. If returning 0 everything is OK, if not returning the error code*)
	VAR_INPUT
		xStackEnabled : BOOL;
	END_VAR
END_FUNCTION

FUNCTION CheckItemInStack : UDINT (*INTERNAL. Check the item is in the Stack when is expected to be*)
	VAR_INPUT
		Id : DINT;
		StackArray : REFERENCE TO ARRAY[0..THICK_MEDIATRACKING_MAX_MEDIA] OF stThicknessCtrl_MediaPosStatus;
		TotalElements : UINT;
	END_VAR
	VAR_IN_OUT
		PositionFound : UINT;
	END_VAR
	VAR
		iIndex : UINT;
	END_VAR
END_FUNCTION

FUNCTION CheckNotItemInStack : UDINT (*INTERNAL. Check the item is NOT in the Stack when is expected NOT to be*)
	VAR_INPUT
		Id : DINT;
		StackArray : REFERENCE TO ARRAY[0..THICK_MEDIATRACKING_MAX_MEDIA] OF stThicknessCtrl_MediaPosStatus;
		TotalElements : UINT;
	END_VAR
	VAR_IN_OUT
		PositionFound : UINT;
	END_VAR
	VAR
		iIndex : UINT;
	END_VAR
END_FUNCTION

FUNCTION AssignItemInStack : UDINT (*INTERNAL. Assignation without any checking if the item is or is not in the array*)
	VAR_INPUT
		ItemMedia : REFERENCE TO stThicknessCtrl_MediaConfig;
		StackArray : REFERENCE TO ARRAY[0..THICK_MEDIATRACKING_MAX_MEDIA] OF stThicknessCtrl_MediaPosStatus;
		Position : UINT; (*The position to insert the element*)
		TotalElementsStack : UINT;
	END_VAR
	VAR
		ItemEnergyFake : stThickCtrl_Energy;
	END_VAR
END_FUNCTION

FUNCTION AssignItemEnergyInStack : UDINT (*INTERNAL. Assignation without any checking if the item is or is not in the array*)
	VAR_INPUT
		ItemMedia : REFERENCE TO stThicknessCtrl_MediaConfig;
		ItemEnergy : REFERENCE TO stThickCtrl_Energy;
		StackArray : REFERENCE TO ARRAY[0..THICK_MEDIATRACKING_MAX_MEDIA] OF stThicknessCtrl_MediaPosStatus;
		EnergyArray : REFERENCE TO ARRAY[0..THICK_MEDIATRACKING_MAX_MEDIA_x2] OF stThickCtrl_Energy;
		PositionStack : UINT; (*The position to insert the element*)
		PositionEnergy : USINT; (*The position to insert the element*)
	END_VAR
END_FUNCTION

FUNCTION AssignLastItemInStack : UDINT (*Check if the Line to stack is correct. If returning 0 everything is OK, if not returning the error code*)
	VAR_INPUT
		ItemMedia : REFERENCE TO stThicknessCtrl_MediaConfig;
		StackArray : REFERENCE TO ARRAY[0..THICK_MEDIATRACKING_MAX_MEDIA] OF stThicknessCtrl_MediaPosStatus;
	END_VAR
	VAR_IN_OUT
		TotalElementsStack : UINT;
	END_VAR
	VAR
		ItemEnergyFake : stThickCtrl_Energy;
		IndexEnergyFake : USINT;
	END_VAR
END_FUNCTION

FUNCTION AssignLastItemEnergyInStack : UDINT (*Check if the Line to stack is correct. If returning 0 everything is OK, if not returning the error code*)
	VAR_INPUT
		ItemMedia : REFERENCE TO stThicknessCtrl_MediaConfig;
		ItemEnergy : REFERENCE TO stThickCtrl_Energy;
		StackArray : REFERENCE TO ARRAY[0..THICK_MEDIATRACKING_MAX_MEDIA] OF stThicknessCtrl_MediaPosStatus;
		EnergyArray : REFERENCE TO ARRAY[0..THICK_MEDIATRACKING_MAX_MEDIA_x2] OF stThickCtrl_Energy;
	END_VAR
	VAR_IN_OUT
		TotalElementsStack : UINT;
		IndexEnergy : USINT;
	END_VAR
	VAR
		PositionFound : UINT;
	END_VAR
END_FUNCTION

FUNCTION InsertItemInStack : UDINT (*Check if the Line to stack is correct. If returning 0 everything is OK, if not returning the error code*)
	VAR_INPUT
		Id : DINT;
		ItemMedia : REFERENCE TO stThicknessCtrl_MediaConfig;
		StackArray : REFERENCE TO ARRAY[0..THICK_MEDIATRACKING_MAX_MEDIA] OF stThicknessCtrl_MediaPosStatus;
	END_VAR
	VAR_IN_OUT
		TotalElementsStack : UINT;
	END_VAR
	VAR
		ItemEnergyFake : stThickCtrl_Energy;
		IndexEnergyFake : USINT;
		PositionFound : UINT;
	END_VAR
END_FUNCTION

FUNCTION InsertItemEnergyInStack : UDINT (*Check if the Line to stack is correct. If returning 0 everything is OK, if not returning the error code*)
	VAR_INPUT
		Id : DINT;
		ItemMedia : REFERENCE TO stThicknessCtrl_MediaConfig;
		ItemEnergy : REFERENCE TO stThickCtrl_Energy;
		StackArray : REFERENCE TO ARRAY[0..THICK_MEDIATRACKING_MAX_MEDIA] OF stThicknessCtrl_MediaPosStatus;
		EnergyArray : REFERENCE TO ARRAY[0..THICK_MEDIATRACKING_MAX_MEDIA_x2] OF stThickCtrl_Energy;
	END_VAR
	VAR_IN_OUT
		TotalElementsStack : UINT;
		IndexEnergy : USINT;
	END_VAR
	VAR
		PositionFound : UINT;
		CheckResult : UDINT;
	END_VAR
END_FUNCTION

FUNCTION RemoveItemInStack : UDINT (*Check if the Line to stack is correct. If returning 0 everything is OK, if not returning the error code*)
	VAR_INPUT
		Id : DINT;
		StackArray : REFERENCE TO ARRAY[0..THICK_MEDIATRACKING_MAX_MEDIA] OF stThicknessCtrl_MediaPosStatus;
	END_VAR
	VAR_IN_OUT
		TotalElementsStack : UINT;
	END_VAR
	VAR
		CheckResult : UDINT;
		PositionFound : UINT;
	END_VAR
END_FUNCTION
```

#### LoadMedia.st
```iecst
(* Loading Fast data in an array to an array of tracking data. Using USINT array to load differente lines *)
FUNCTION LoadMediaFromFastDataLine

	//Creating mask with bit active in the right position
	bitLine:=1;
	bitLine := SHL(bitLine,indexLine);

	IF REAL_TO_UINT(fastValues) >= positionsToRunArray THEN
		// More values than holes to fill-in. Distribution of data. If there is a gap in the Fast Data, the gap has to appear in the slow data
		rValuesPerPosition :=  fastValues / UINT_TO_REAL(positionsToRunArray);
		FOR iIndexArray:=0 TO positionsToRunArray -1 DO
			//Activate the bit
			valuesTracking[iIndexArray + sensorPosition] := valuesTracking[iIndexArray + sensorPosition] OR bitLine;
			// If MOD is 0, no need to wonder about TRUNC or CEIL
			IF brmfmod(fastValues, UINT_TO_REAL(positionsToRunArray)) = 0 THEN
				iFirstIndex := REAL_TO_UINT(UINT_TO_REAL(iIndexArray) * rValuesPerPosition);
				FOR iIndexNewMediaArray := iFirstIndex TO iFirstIndex + REAL_TO_UINT(rValuesPerPosition) -1 DO
					IF NOT newValues[iIndexNewMediaArray] THEN
						//Resetting the bit
						valuesTracking[iIndexArray + sensorPosition] := valuesTracking[iIndexArray + sensorPosition] AND NOT(bitLine);
					END_IF
				END_FOR
			ELSE
				FOR iIndexNewMediaArray := INT_TO_UINT(TRUNC(UINT_TO_REAL(iIndexArray) * rValuesPerPosition)) TO MIN(INT_TO_UINT(TRUNC(UINT_TO_REAL(iIndexArray + 1) * rValuesPerPosition )), REAL_TO_UINT(fastValues -1)) DO
					IF NOT newValues[iIndexNewMediaArray] THEN
						//Resetting the bit
						valuesTracking[iIndexArray + sensorPosition] := valuesTracking[iIndexArray + sensorPosition] AND NOT(bitLine);
					END_IF
				END_FOR
			END_IF
		END_FOR
	ELSE
		// More holes than data. Ampliation of data
		rValuesPerPosition :=  fastValues / UINT_TO_REAL(positionsToRunArray);
		FOR iIndexArray :=0 TO positionsToRunArray -1 DO
			iFirstIndex := INT_TO_UINT(TRUNC(UINT_TO_REAL(iIndexArray) * rValuesPerPosition));
			iLastIndex := MIN(INT_TO_UINT(TRUNC(UINT_TO_REAL(iIndexArray +1 ) * rValuesPerPosition )), REAL_TO_UINT(fastValues-1));
			FOR iIndexNewMediaArray := iFirstIndex TO iLastIndex DO
				IF newValues[iIndexNewMediaArray] THEN
					//Activate the bit
					valuesTracking[iIndexArray + sensorPosition] := valuesTracking[iIndexArray + sensorPosition] OR bitLine;
				ELSE
					//Reset the bit
					valuesTracking[iIndexArray + sensorPosition] := valuesTracking[iIndexArray + sensorPosition] AND NOT(bitLine);
				END_IF
			END_FOR
		END_FOR
	END_IF

	LoadMediaFromFastDataLine := TRUE;
	valuesTracking; // To monitor while debugging

END_FUNCTION

(* Loading Fast data in an array to an array of tracking data. Using BOOL array to load individual data *)
FUNCTION LoadMediaFromFastDataBool

	IF REAL_TO_UINT(fastValues) >= positionsToRunArray THEN
		// More values than holes to fill-in. Distribution of data. If there is a gap in the Fast Data, the gap has to appear in the slow data
		rValuesPerPosition :=  fastValues / UINT_TO_REAL(positionsToRunArray);
		FOR iIndexArray:=0 TO positionsToRunArray -1 DO
			//Activate the bit
			valuesTracking[iIndexArray + sensorPosition] := TRUE;
			// If MOD is 0, no need to wonder about TRUNC or CEIL
			IF brmfmod(fastValues, UINT_TO_REAL(positionsToRunArray)) = 0 THEN
				iFirstIndex := REAL_TO_UINT(UINT_TO_REAL(iIndexArray) * rValuesPerPosition);
				FOR iIndexNewMediaArray := iFirstIndex TO iFirstIndex + REAL_TO_UINT(rValuesPerPosition) -1 DO
					IF NOT newValues[iIndexNewMediaArray] THEN
						//Resetting the bit
						valuesTracking[iIndexArray + sensorPosition] := FALSE;
					END_IF
				END_FOR
			ELSE
				FOR iIndexNewMediaArray := INT_TO_UINT(TRUNC(UINT_TO_REAL(iIndexArray) * rValuesPerPosition)) TO MIN(INT_TO_UINT(TRUNC(UINT_TO_REAL(iIndexArray + 1) * rValuesPerPosition )), REAL_TO_UINT(fastValues -1)) DO
					IF NOT newValues[iIndexNewMediaArray] THEN
						//Resetting the bit
						valuesTracking[iIndexArray + sensorPosition] := FALSE;
					END_IF
				END_FOR
			END_IF
		END_FOR
	ELSE
		// More holes than data. Ampliation of data
		rValuesPerPosition :=  fastValues / UINT_TO_REAL(positionsToRunArray);
		FOR iIndexArray :=0 TO positionsToRunArray -1 DO
			iFirstIndex := INT_TO_UINT(TRUNC(UINT_TO_REAL(iIndexArray) * rValuesPerPosition));
			iLastIndex := MIN(INT_TO_UINT(TRUNC(UINT_TO_REAL(iIndexArray +1 ) * rValuesPerPosition )), REAL_TO_UINT(fastValues-1));
			FOR iIndexNewMediaArray := iFirstIndex TO iLastIndex DO
				valuesTracking[iIndexArray + sensorPosition] := newValues[iIndexNewMediaArray];
			END_FOR
		END_FOR
	END_IF
	LoadMediaFromFastDataBool := TRUE;

END_FUNCTION
```

#### ReviewTracking.st
```iecst
(* Review if any element in the array is inside de window *)
FUNCTION ReviewMediaTrackingInPosition

	// If no elements inside, return
	IF TotalElementsInside = 0 THEN
		ReviewMediaTrackingInPosition := FALSE;
		RETURN;
	END_IF

	xMediaInPosition := FALSE;
	FOR iIndexArray := 0 TO TotalElementsInside - 1 DO
		IF NOT xIsWhite OR ArrayOfMedia[iIndexArray].Media.xHasWhite THEN
			IF ArrayOfMedia[iIndexArray].HeadPosition < iStartWindow THEN
				// Waiting the media
			ELSIF ArrayOfMedia[iIndexArray].HeadPosition >= iStartWindow AND ArrayOfMedia[iIndexArray].HeadPosition <= iEndWindow THEN
				xMediaInPosition := TRUE;
			ELSIF ArrayOfMedia[iIndexArray].HeadPosition > iEndWindow THEN
				xMediaInPosition := ArrayOfMedia[iIndexArray].TailPosition <= iEndWindow;
			END_IF
		END_IF
	END_FOR
	ReviewMediaTrackingInPosition := xMediaInPosition;

END_FUNCTION

(* Review if any element in the array is inside de window and calculate the Energy needed *)
FUNCTION RevMediaTrackingEnergyInPos

	// If no elements inside, return
	IF TotalElementsInside = 0 THEN
		RevMediaTrackingEnergyInPos := FALSE;
		RETURN;
	END_IF

	// If more lamps than configured, return
	IF iTotalLamps > THICKENERGY_MAX_LAMPS THEN
		RevMediaTrackingEnergyInPos := FALSE;
		RETURN;
	END_IF

	// Reset Energy Values
	FOR iIndexArray := 0 TO iTotalLamps - 1 DO
		Intensity[iIndexArray] := 0;
	END_FOR

	FOR iIndexArray := 0 TO TotalElementsInside - 1 DO

		diPosStartMedia := ArrayOfMedia[iIndexArray].HeadPosition;
		diPosEndMedia := UDINT_TO_DINT(ArrayOfMedia[iIndexArray].HeadPosition) - REAL_TO_DINT(ArrayOfMedia[iIndexArray].Media.rLength/10);

		IF diPosStartMedia >= INT_TO_DINT(iStartWindow) AND diPosEndMedia <= INT_TO_DINT(iEndWindow) THEN

			// If no proper pointer, return to avoid a crash
			IF ArrayOfMedia[iIndexArray].pMediaEnery = 0 THEN
				RevMediaTrackingEnergyInPos := FALSE;
				RETURN;
			END_IF

			RevMediaTrackingEnergyInPosItem(ADR(ArrayOfMedia[iIndexArray]), ArrayOfMedia[iIndexArray].pMediaEnery ,iStartWindow, iEndWindow, rLampWidth, rLampOffset, rLampOverlap, Intensity);

		END_IF

	END_FOR

	// Asign data to received array. iIntensity starsts in 1
	FOR iIndexArray := 1 TO iTotalLamps DO
		iIntensity[iIndexArray] := MAX(Intensity[iTotalLamps - iIndexArray], iMinIntensity);
	END_FOR

	RevMediaTrackingEnergyInPos := TRUE;

	Intensity; // INTERNAL variable. To monitor
	iIntensity; // IN_OUT variable. To monitor

END_FUNCTION

(* Review if any element in the array is inside de window and calculate the Energy needed *)
FUNCTION RevMediaTrackingEnergyInPosItem

	//   The first LAMP is in the operator side, but for easier calculations, in this point the arrays will have the
	// same order as the information in the document. Later, the array will be swapped to send it to Dryer

	rOffsetStartDocument := MediaData.Media.rCrossOffset;

	iFirstLamp := INT_TO_UINT(MAX(0,TRUNC((rOffsetStartDocument - rLampOffset)/rLampWidth)));
	iLastLamp := INT_TO_UINT(LIMIT(0,TRUNC((rOffsetStartDocument + MediaData.Media.rWidth - rLampOffset)/rLampWidth), THICKENERGY_MAX_LAMPS-1));

	(* Calculus explanation to get First and Last section to avoid loop a for over the array

		iFirstCrossSection is where: PosEndSection_i > PosIniLamp_j
		iLastCrossSection is where: PosIniSection_i < PosEndLamp_j
	*)

	iFirstProcessSection := LIMIT(0,REAL_TO_INT(TRUNC(UDINT_TO_REAL(MediaData.HeadPosition - iEndWindow))/THICKENERGY_PROCESS_STEP), THICKENERGY_MAX_PROCESS_ITEMS);
	iLastProcessSection := LIMIT(0,REAL_TO_INT(TRUNC(UDINT_TO_REAL(MediaData.HeadPosition - iStartWindow))/THICKENERGY_PROCESS_STEP),THICKENERGY_MAX_PROCESS_ITEMS);

	FOR iIndexLamp := iFirstLamp TO iLastLamp DO
		iLampIntensity := 0;

		(* Calculus explanation to get First and Last section to avoid loop a for over the array

		PosIniSection_i = rOffsetStartDocument + THICKENERGY_CROSS_STEP * i
		PosEndSection_i = rOffsetStartDocument + THICKENERGY_CROSS_STEP * (i +1)
		PosIniLamp_j = rLampOffset + rLampWidth * j
		PosEndLamp_j = rLampOffset + rLampWidth * (j +1)

		*)

		iFirstCrossSection := LIMIT(0, REAL_TO_INT(MAX(0,brmceil(((rLampOffset + rLampWidth * iIndexLamp - rOffsetStartDocument - rLampOverlap)/ THICKENERGY_CROSS_STEP)-1))), THICKENERGY_MAX_CROSS_ITEMS);
		iLastCrossSection := LIMIT(0, REAL_TO_INT(TRUNC(((rLampOffset + rLampWidth * (iIndexLamp + 1) - rOffsetStartDocument + rLampOverlap)/ THICKENERGY_CROSS_STEP))), THICKENERGY_MAX_CROSS_ITEMS);

		FOR iIndexCross := iFirstCrossSection TO iLastCrossSection DO

			FOR iIndexProcess := iFirstProcessSection TO iLastProcessSection DO
				iLampIntensity := MAX(iLampIntensity, EnergyData.iPower[iIndexProcess,iIndexCross]);
			END_FOR

		END_FOR
		iIntensity[iIndexLamp] := MAX(iIntensity[iIndexLamp], iLampIntensity);

	END_FOR

	RevMediaTrackingEnergyInPosItem := TRUE;

END_FUNCTION
```

#### CheckStack.st
```iecst
FUNCTION CheckMediaToStack

	CheckMediaToStack := 0;

	IF CheckEnabledStack(xStackEnabled) > 0 THEN
		CheckMediaToStack := CheckEnabledStack(xStackEnabled);
		RETURN;
	END_IF

	IF CheckLineToStack(NewMedia.iLine, xStackEnabled, xDtpEnabled) > 0 THEN
		CheckMediaToStack := CheckLineToStack(NewMedia.iLine, xStackEnabled, xDtpEnabled);
		RETURN;
	END_IF

	IF NewMedia.rThickness < 0.1 OR NewMedia.rThickness > rMaxThickness THEN
		CheckMediaToStack := 160; // Thickness error
		RETURN;
	END_IF

	IF NewMedia.rWidth < rMinWidth OR NewMedia.rWidth > rMaxWidth THEN
		CheckMediaToStack := 170; // Width error
		RETURN;
	END_IF

	IF NewMedia.rLength < rMinLength OR NewMedia.rLength > rMaxLength THEN
		CheckMediaToStack := 180; // Length error
		RETURN;
	END_IF

	//	IF NewMedia.rGap < 10 THEN
	//		CheckMediaToStack := 190; // Gap error
	//		RETURN;
	//	END_IF

	IF NewMedia.rCrossOffset < -NewMedia.rWidth/2 OR (NewMedia.rWidth + NewMedia.rCrossOffset) > rMaxWidth/2 THEN
		CheckMediaToStack := 200; // Offset error
		RETURN;
	END_IF

	IF NewMedia.rDocWidth < 0 OR NewMedia.rDocWidth > NewMedia.rWidth THEN
		CheckMediaToStack := 210; // DocWidth error
		RETURN;
	END_IF

	IF NewMedia.rDocLength < 0 OR NewMedia.rDocLength > NewMedia.rLength THEN
		CheckMediaToStack := 220; // DocLength error
		RETURN;
	END_IF

	IF NewMedia.rDocCrossOffset < -NewMedia.rWidth/2 OR (NewMedia.rDocWidth + NewMedia.rDocCrossOffset) > rMaxWidth/2 THEN
		CheckMediaToStack := 230; // DocCrossOffset error
		RETURN;
	END_IF

	IF NewMedia.rDocProcessOffset < 0 OR (NewMedia.rDocLength + NewMedia.rDocProcessOffset) > NewMedia.rDocLength THEN
		CheckMediaToStack := 240; // DocProcessOffset error
		RETURN;
	END_IF

	IF NewMedia.iLine = 1 AND xStackLine1Full THEN
		CheckMediaToStack := 500; // Array full
		RETURN;
	END_IF

	IF NewMedia.iLine = 2 AND xStackLine2Full THEN
		CheckMediaToStack := 501; // Array full
		RETURN;
	END_IF

END_FUNCTION

FUNCTION CheckLineToStack

	CheckLineToStack := 0;

	IF CheckEnabledStack(xStackEnabled) > 0 THEN
		CheckLineToStack := CheckEnabledStack(xStackEnabled);
		RETURN;
	END_IF

	IF NOT xDtpEnabled THEN
		IF iLine <> 1 THEN
			CheckLineToStack := 150; // Line error
			RETURN;
		END_IF
	ELSE
		IF iLine < 1 OR iLine > 2 THEN
			CheckLineToStack := 150; // Line error
			RETURN;
		END_IF
	END_IF

END_FUNCTION

FUNCTION CheckEnabledStack

	CheckEnabledStack := 0;

	IF NOT xStackEnabled THEN
		CheckEnabledStack := 140; // Stack not enabled
		RETURN;
	END_IF

END_FUNCTION

FUNCTION CheckItemInStack

	CheckItemInStack := 0;

	// Check if the Id is valid
	IF Id < 0 THEN
		CheckItemInStack := 1500; // Id negative. Not in Array
		RETURN;
	END_IF

	// If not elements, the Id is not in list
	IF TotalElements = 0 THEN
		CheckItemInStack := 1510; // Id Not found in Array
		RETURN;
	END_IF

	// Check if the id is in the array
	FOR iIndex := 0 TO TotalElements - 1 DO
		IF Id = StackArray[iIndex].Media.id THEN
			CheckItemInStack := 0; // Id Found
			PositionFound := iIndex; // Returning the position where Id is
			RETURN;
		END_IF
	END_FOR

	// The id has not been found. Raise an error
	CheckItemInStack := 1510; // Id Not found in Array
	RETURN;

END_FUNCTION

FUNCTION CheckNotItemInStack

	CheckNotItemInStack := 0;

	// Check if the Id is valid
	IF Id < 0 THEN
		CheckNotItemInStack := 1500; // Id negative. Not in Array
		RETURN;
	END_IF

	// If not elements, the Id is not in list
	IF TotalElements = 0 THEN
		CheckNotItemInStack := 0; // Id Not found in Array
		RETURN;
	END_IF

	// Check if the id is in the array
	FOR iIndex := 0 TO TotalElements - 1 DO
		IF Id = StackArray[iIndex].Media.id THEN
			CheckNotItemInStack := 1520; // Id FOUND in Array
			PositionFound := iIndex; // Returning the position where Id is
			RETURN;
		END_IF
	END_FOR

END_FUNCTION
```

### Package Logical/ExtPack/_Media/ThicknessCtrl/ThicknessCtrl_v2 - Heigt detection and empty belt logic

### ThicknessCtrl.typ
```iecst
TYPE
	ThicknessCtrl_RejectBoardEdge :
		(
		REJECT_FRONT,
		REJECT_REAR
		);
	stThicknessCtrl_ouputs_typ : 	STRUCT  (*For now just a copy of ALL parameters*)
		xHoldReject : BOOL; (*While signal is active, reject remains activated*)
		xReject : BOOL; (*Signal for stacker to reject a single board*)
		xEnableMediaSignalToCb : BOOL;
		xMediaFiltered : BOOL; (*Signal active when detection system detects a real media*)
	END_STRUCT;
	stThicknessCtrl_CheckMediaInput : 	STRUCT
		xCheckFail : BOOL; (*Media is not detected when it sould be*)
	END_STRUCT;
	stThicknessCtrl_inputs_typ : 	STRUCT  (*For now just a copy of ALL parameters*)
		xVirtualMedia : BOOL; (*Virtual Media Present a the entrance of the machine (Instant or Continuous print)*)
		CheckMedia : ARRAY[0..MAX_LAST_CHECKMEDIA]OF stThicknessCtrl_CheckMediaInput;
	END_STRUCT;
	stThickCtrl_StackStatus_typ : 	STRUCT  (*For now just a copy of ALL parameters*)
		iInsideMediaL1 : USINT; (*Total media below the blocks*)
		iInsideMediaL2 : USINT; (*Total media below the blocks*)
		iNewMediaLoadedL1 : UINT; (*Total new media loaded*)
		iNewMediaLoadedL2 : UINT; (*Total new media loaded*)
	END_STRUCT;
	stThickCtrl_HeighStatus_typ : 	STRUCT  (*For now just a copy of ALL parameters*)
		iMediaHeigh : UINT; (*Value measured of the media heigh in mm (max 650mm, resolution 0.01)*)
		rMediaHeigh : REAL; (*Value measured of the media heigh in mm (max 650mm)*)
		rMediaThickness : REAL; (*Value of the expected Thickness value depending on the configuration of the machine. ContinuousMedia or from Stack*)
		rMediaThicknessMargin : REAL; (*Value of the expected Thickness+Margin value depending on the configuration of the machine. ContinuousMedia or from Stack*)
		xIncreasedHeigh : ARRAY[0..TOTAL_THICKNESS_SECTIONS]OF BOOL;
		rMaxHeigh : ARRAY[0..TOTAL_THICKNESS_SECTIONS]OF REAL; (*Valuen in mm  NOTE: Element 0 is not used*)
	END_STRUCT;
	stThickCtrl_RejectStatus_typ : 	STRUCT  (*For now just a copy of ALL parameters*)
		xRejecting : BOOL; (*Active when reject is activated. This signal is a 2 secons pulse to allow see it*)
		iBoardsRejected : UINT; (*Counter of boards rejected by stacker*)
		iTimesInRejection : UINT; (*Counter of boards rejected*)
		iTimesInRejectionToday : UINT; (*Counter of boards rejected*)
	END_STRUCT;
	stThickCtrl_DetSystemStatus_typ : 	STRUCT  (*For now just a copy of ALL parameters*)
		xInPosition : BOOL; (*Active when device used for thicknessctrl is positioned for printing*)
	END_STRUCT;
	stThickCtrl_BeltStatus_typ : 	STRUCT  (*For now just a copy of ALL parameters*)
		xBeltEmpty : BOOL;
		iBeltTurns : UINT;
		rBeltPositionMmInit : REAL;
		rBeltPositionMmFinal : REAL;
		rBeltSpeed : REAL;
	END_STRUCT;
	stThickCtrl_DryerIntensityStatus : 	STRUCT
		Intensity : ARRAY[0..THICKENERGY_MAX_LAMPS]OF INT; (*Data starting in index 1*)
	END_STRUCT;
	stThickCtrl_DryerMediaStatus : 	STRUCT
		xMediaInPosition : BOOL;
		Intensity : ARRAY[0..THICKENERGY_MAX_LAMPS]OF INT; (*Data starting in index 1*)
	END_STRUCT;
	stThickCtrl_LedLineMediaStatus : 	STRUCT
		xMediaInLedPosition : BOOL;
		Media : stThicknessCtrl_MediaConfig;
	END_STRUCT;
	stThickCtrl_LineMediaStatus : 	STRUCT
		White : stThickCtrl_LedLineMediaStatus;
		Color : stThickCtrl_LedLineMediaStatus;
		Primer : stThickCtrl_LedLineMediaStatus;
		NirDryer : ARRAY[0..MAX_LAST_NIR_MODULES]OF stThickCtrl_DryerMediaStatus;
		InsideMedia : ARRAY[0..THICK_MEDIATRACKING_MAX_MEDIA]OF stThicknessCtrl_MediaPosStatus;
		iBoardsBelowBlock : UINT; (*Counter of boards that are below the printer properly detected by productDetect*)
		xDetectionSystemIncoherence : BOOL; (*There is no media detection consistensy between PD an the array sensor*)
	END_STRUCT;
	stThickCtrl_MediaPositionStatus : 	STRUCT  (*For now just a copy of ALL parameters*)
		xMediaAtPrinterExit : BOOL; (*There is media at the end of printer's belt*)
		xMediaInside : BOOL; (*Some media has passed the first sensor and still not exited*)
		xTrackingEmpty : BOOL; (*Some media has passed the first sensor and still not exited the tracking distance*)
		xMountedMediaInside : BOOL;
		xVirtualMediaInside : BOOL; (*Some Virtual media has passed the first sensor and still not exited*)
		xMediaToRejectInside : BOOL; (*Media to be rejected has beed detected and it is below the machine*)
		xMediaBelowMachine : BOOL; (*There is media below the machine (not considered the distance between the sensor and the first block)*)
		xMediaInWarpSensorPosition : BOOL;
		L1 : stThickCtrl_LineMediaStatus;
		L2 : stThickCtrl_LineMediaStatus;
		iBoardsBelowBlock : UINT; (*Counter of boards that are below the printer properly detected by productDetect*)
	END_STRUCT;
	stThickCtrl_DetectionStatus_typ : 	STRUCT  (*For now just a copy of ALL parameters*)
		xMediaInProductDetect : BOOL;
		xMediaToRejectDetected : BOOL; (*Media to be rejected is beed detected now*)
		xFilteredProductDetectMediaL1 : BOOL;
		xFilteredProductDetectMediaL2 : BOOL;
		xFilteredAnalogSensorMedia : BOOL;
		xFilteredArraySensorMedia : BOOL;
		xFilteredBasicDetectionMedia : BOOL;
		iBoardsFromStartL1 : UDINT; (*Detected boards since belt is started. Reseted when belt starts again. Needed media tracking enable to use it*)
		iBoardsFromStartL2 : UDINT; (*Detected boards since belt is started. Reseted when belt starts again. Needed media tracking enable to use it*)
		iTotalBoardsL1 : UDINT; (*Detected boards since PLC is started. Needed media tracking enable to use it*)
		iTotalBoardsL2 : UDINT; (*Detected boards since PLC is started. Needed media tracking enable to use it*)
	END_STRUCT;
	stThicknessCtrl_status_typ : 	STRUCT  (*For now just a copy of ALL parameters*)
		Detection : stThickCtrl_DetectionStatus_typ;
		MediaPosition : stThickCtrl_MediaPositionStatus;
		Belt : stThickCtrl_BeltStatus_typ;
		DetectionSystem : stThickCtrl_DetSystemStatus_typ;
		Dry : ARRAY[0..MAX_LAST_NIR_MODULES]OF stThickCtrl_DryerIntensityStatus;
		Reject : stThickCtrl_RejectStatus_typ;
		Heigh : stThickCtrl_HeighStatus_typ;
		Stack : stThickCtrl_StackStatus_typ;
		iReadEnergyFileStep : USINT; (*1: Idle, 255:Error*)
		xNewMediaStackEnabled : BOOL; (*New Media Stack functionality enabled in the PLC*)
		xMediaTrackingEnabled : BOOL; (*Media Tracking functionality enabled in the PLC*)
	END_STRUCT;
	ThicknessCtrl_PositionSect_typ : 	STRUCT  (*Structure to define the position to detect if there is media below*)
		iPosition : UINT; (*Value in cm from the sensor*)
	END_STRUCT;
	stThicknessCtrl_Section_typ : 	STRUCT
		iEnd : UINT;
		iStart : UINT;
		xEnabled : BOOL := FALSE;
	END_STRUCT;
	stThicknessCtrl_BeltParams : 	STRUCT
		iBeltPerimeterLength : UINT; (*Perimeter of belt. Value in cm*)
		rMinBeltSpeedToStart : REAL; (*Value of the Speed in m/min*)
		iDistanceEmptyBeltIni : INT; (*Distance in cm from thickness media sensor detector to the end of the belt. This distance is mechanical. Not related with Reject*)
		rBeltSpeed : REAL; (*Current Belt Speed in m/min*)
	END_STRUCT;
	stThicknessCtrl_RejectParams : 	STRUCT
		iHoldRejectDistance : INT; (*Distance between end of printer's belt and stacker's hold reject position in cm. If negative, the reject signal is given with the media inside the printer*)
		iRejectDistance : INT; (*Distance between end of printer's belt and stacker's reject sheet position in cm. If negative, the reject signal is given with the media inside the printer*)
		RejectBoardEdge : ThicknessCtrl_RejectBoardEdge; (*Reject the boards with the FrontEdge or with the RearEdge*)
		xRejectTracking : BOOL; (*Reject feature active and reject array has to be evaluated*)
		xLoadMediaFromProductDetect : BOOL; (*Source of the media data*)
	END_STRUCT;
	stThickCtrl_SecDetectionParams : 	STRUCT
		iMediaFilter : UINT;
		iSensorPosition : UINT; (*Position of the sensor in X direction in cm*)
		xLoadMedia : BOOL; (*Source of the media data*)
		xEnableMediaTracking : BOOL; (*Track the data of the sensor in the present media array*)
		xEnableSensorIncoherAlarm : BOOL; (*Enable the sensor incoherenci alarm, reviewing the sensor array in detection when arriving media to ProductDetect*)
	END_STRUCT;
	stThickCtrl_DetectionPrDetPar : 	STRUCT
		iMediaFilter : UINT;
		iSensorPosition : UINT; (*Position of the sensor in X direction in cm*)
		xLoadMedia : BOOL; (*Source of the media data*)
		xFixedSensor : BOOL; (*Active if the sensor is fixed and reads properly always*)
		pMediaInProductDetectL1 : {REDUND_UNREPLICABLE} UDINT; (*Pointer to MediaInProductDetect*)
		pMediaInProductDetectL2 : {REDUND_UNREPLICABLE} UDINT; (*Pointer to MediaInProductDetect*)
	END_STRUCT;
	stThicknessCtrl_DetectionParams : 	STRUCT
		ProductDetect : stThickCtrl_DetectionPrDetPar;
		Array : stThickCtrl_SecDetectionParams;
		Analog : stThickCtrl_SecDetectionParams;
		Basic : stThickCtrl_SecDetectionParams;
		xEnabledStack : BOOL; (*Use the stack for considering the new media is entering the machine. If disabled, new media taken from continuous media*)
	END_STRUCT;
	stThicknessCtrl_NirDryerParams : 	STRUCT
		iPosition : UINT; (*Center position of the Dryer*)
	END_STRUCT;
	stThicknessCtrl_CureLampParams : 	STRUCT
		iStartWindow : UINT; (*Initial position of curing window in cm*)
		iEndWindow : UINT; (*End position of curing window in cm*)
		xEnabled : BOOL; (*Enabled to cure*)
	END_STRUCT;
	stThicknessCtrl_CureParams : 	STRUCT
		xEnableTracking : BOOL; (*Cure feature active and reject array has to be evaluated. OLD ARRAY IMPLEMENTATION*)
		xEnableMediaTracking : BOOL; (*Cure MediaTracking is activated and has to be evaluated*)
		White : stThicknessCtrl_CureLampParams;
		Color : stThicknessCtrl_CureLampParams;
		Primer : stThicknessCtrl_CureLampParams;
	END_STRUCT;
	stThicknessCtrl_NirDryParams : 	STRUCT
		xDryStack : BOOL; (*Use the stack for considering the new media is entering the machine. If disabled, new media taken from continuous media*)
		xEnableMediaTracking : BOOL; (*Dry tracking is activated and has to be evaluated*)
		rCommsDelay : REAL; (*Comms delay in ms*)
		rThermalDelay : REAL; (*Thermal delay in ms*)
		rSubstratePowerReduction : REAL := 1.0; (*Substrate power reduction. From 1.0 (default) to 0.3 is allowed*)
		rThermalInerciaReduction : REAL := 1.0; (*Thermal Inercia Power reduction. From 1.0 (default) to 0.8 is allowed*)
		iMinDryValue : INT; (*Minimum value to consider when no media is detected. To avoid sending 0 and the change is too big*)
		iLamps : USINT; (*Total quantity of Lamps in the machine*)
		rLampWidth : REAL := 30; (*Width of each lamp. Value in mm*)
		rLampOffset : REAL := 700; (*Offset of the LAST  lamp considering the center of the belt as 0. Positive to operator side. Value in mm*)
		rDryExtend : REAL := 0; (*Extra width to consider for each lamp in each side to check the image to dry. Value in mm*)
		Dryers : ARRAY[0..MAX_LAST_NIR_MODULES]OF stThicknessCtrl_NirDryerParams;
	END_STRUCT;
	stThicknessCtrl_CheckMediaParams : 	STRUCT
		xActive : BOOL; (*Activate CheckMedia. If media should be there but there is not, raise a signa to define an alarm*)
		xCheckGap : BOOL; (*Activate Checking the gap after the Media. This should just be activated if the machine ALWAYS have a quite big gap between media*)
		CheckPosition : UINT; (*Position of the sensor to check the media should be there. Value in cm*)
		CheckDelayPosition : UINT; (*Positions of the sensor to wait to be inside the board. Value in cm*)
		iSensorFilter : REAL; (*Distance with the signal activated/deactivated to consider the value of the sensor has changed. Value in mm*)
	END_STRUCT;
	stThicknessCtrl_params_typ : 	STRUCT
		AutoMode : stEFI_MachineAutoModes; (*Machine modes operate in automatic mode*)
		Mode : StGeneral_States_Mode; (*Machine general modes (manual, zero, automatic)*)
		iTotalBlocksLengh : UINT; (*Value in cm*)
		Detection : stThicknessCtrl_DetectionParams;
		Cure : stThicknessCtrl_CureParams;
		Dry : stThicknessCtrl_NirDryParams;
		CheckMedia : ARRAY[0..MAX_LAST_CHECKMEDIA]OF stThicknessCtrl_CheckMediaParams; (*CheckMedia to detect jams. 0 not used*)
		Belt : stThicknessCtrl_BeltParams;
		xDoubleLine : BOOL; (*Double line active*)
		sections : ARRAY[0..TOTAL_THICKNESS_SECTIONS]OF stThicknessCtrl_Section_typ;
		iSections : USINT := 1; (*Total quantity of sections used in the machine*)
		Reject : stThicknessCtrl_RejectParams;
		xBlockInProperPrintingPosition : BOOL; (*While block is not in proper position, PD signals going TO CBs are disabled and the boards are rejected*)
		ContinuousMedia : stThickCtrl_EnergyMedia;
		pExtContMedia : UDINT; (*Pointer to stThicknessCtrl_MediaConfig*)
		rMarginSafePrint : REAL; (*Coming from Sw. Fix offset to bent tile. The heads go to the thickness measured + this value. Value in mm*)
		xMarginForBendTile : BOOL; (*To apply margin safe print when photocells installed*)
		rSafetyMarginToHeight : REAL; (*Margin Height  to add to current value in Height array with  commands.xAddSafetyMarginToHeight. Value in mm*)
		rMountedMediaHeigh : REAL; (*Heigh to assign to the rHeigh array when a mounted media is detected*)
		iDistanceFromArrayToPd : UINT; (*Distance from sensor used as reference in array sensor assembly to product detect in process direction*)
		xBlockInPrint : BOOL; (*Block in position state BLOCKP_IN_PRINT*)
	END_STRUCT;
	stThicknessCtrl_paraSw : 	STRUCT
		Dry : stThicknessCtrl_paraSwDry;
	END_STRUCT;
	stThicknessCtrl_paraSwDry : 	STRUCT
		xForceManIntensity : BOOL;
		xReadFile : BOOL; (*Read file from FTP server*)
		xGetMaxFromFileInfo : BOOL; (*When RaiseEdge, clean max data and with RaiseEdge of EmptyBelt, copy max to parSw.Dry.Intensity*)
		ManIntensity : ARRAY[0..MAX_LAST_NIR_MODULES]OF stThickCtrl_DryerIntensityStatus;
	END_STRUCT;
	stThicknessCtrl_Commands_typ : 	STRUCT
		UpdateAllMatrix : BOOL; (*Order to update all the position array just with an edge*)
		xResetMediaBelow : BOOL; (*Reset counters of media below the machine*)
		xRushProof : BOOL; (*Signal from SW to reject media present at the entrance of the machine*)
		xCameraDefectDetected : BOOL; (*Signal from camera to reject media*)
		xAllowToSetMountedMediaHeigh : BOOL; (*Command to let bars to be raised to predefined mounted media heigh position when mounted media alarm*)
		xAddSafetyMarginToHeight : BOOL; (*Command to add the Safety Margin to current Height in the array*)
		xErrorRst : BOOL; (*Order to reset Alarms*)
		xMute : BOOL; (*Mute Order*)
		xReviewIncoherenceArrayAndPd : BOOL;
	END_STRUCT;
	stThicknessCtrl_Orders_typ : 	STRUCT
		xDiscardAllMedia : BOOL; (*Order to discard all media below printer*)
	END_STRUCT;
	stThicknessCtrl_Alarms_typ : 	STRUCT
		xNoThicknessInstalled : BOOL; (*No Thickness System Installed or Selected in SW*)
		CheckMedia : ARRAY[0..MAX_LAST_CHECKMEDIA]OF BOOL; (*0 is not used. Summary of the head and tail alarms*)
		CheckMediaHead : ARRAY[0..MAX_LAST_CHECKMEDIA]OF BOOL; (*0 is not used*)
		CheckMediaTail : ARRAY[0..MAX_LAST_CHECKMEDIA]OF BOOL; (*0 is not used*)
	END_STRUCT;
	stThicknessCtrl_Internal_typ : 	STRUCT
		ProductDetectValuesL1 : ARRAY[0..THICK_MAX_UPDATE_VALUES]OF BOOL; (*Values of the digital signal. 0 is not used*)
		ProductDetectValuesL2 : ARRAY[0..THICK_MAX_UPDATE_VALUES]OF BOOL; (*Values of the digital signal. 0 is not used*)
		MediaArraySensorValues : ARRAY[0..THICK_MAX_UPDATE_VALUES]OF BOOL; (*Values of the digital signal. 0 is not used*)
		MediaAnalogValues : ARRAY[0..THICK_MAX_UPDATE_VALUES]OF BOOL; (*Values of the digital signal. 0 is not used*)
		MediaDetectionValues : ARRAY[0..THICK_MAX_UPDATE_VALUES]OF BOOL; (*Values of the digital signal. 0 is not used*)
		MediaDetectionValuesL1 : ARRAY[0..THICK_MAX_UPDATE_VALUES]OF BOOL; (*Values of the digital signal. 0 is not used*)
		MediaDetectionValuesL2 : ARRAY[0..THICK_MAX_UPDATE_VALUES]OF BOOL; (*Values of the digital signal. 0 is not used*)
		ArrayHeightValues : ARRAY[0..THICK_MAX_UPDATE_VALUES]OF UINT; (*Values of the Thickness Detection signal. 0 is not used*)
		AnalogHeightValues : ARRAY[0..THICK_MAX_UPDATE_VALUES]OF UINT; (*Values of the Thickness Detection signal. 0 is not used*)
		CheckMediaFilteredSensors : ARRAY[0..MAX_LAST_CHECKMEDIA]OF BOOL; (*Filtered signal of the CheckMedia Inputs. 0 not used*)
		rCycleSlow : REAL;
		rCycleFast : REAL;
		iFastValues : UINT; (*Quantity of values read by the fast section of the code each time the slow section is executed*)
		rFastValues : REAL; (*Quantity of values read by the fast section of the code each time the slow section is executed*)
		xMediaToRejectTreated : BOOL;
		rMarginSafePrintChecked : REAL; (*Fix offset to bent tile. The heads go to the thickness measured + this value. Value in mm. Checked minimum value*)
		pMediaTracking : UDINT; (*Pointer to xMediaTracking >> USINT[0..iMAXTRACKINGARRAY]*)
		pDistanceWorkEmptyBelt : UDINT; (*Pointer to iDistanceWorkEmptyBelt*)
		iTotalBoards : UDINT; (*Total boards managed*)
	END_STRUCT;
	stThicknessCtrl_typ : 	STRUCT
		Commands : stThicknessCtrl_Commands_typ;
		Orders : stThicknessCtrl_Orders_typ;
		Inputs : stThicknessCtrl_inputs_typ;
		status : stThicknessCtrl_status_typ;
		parameters : stThicknessCtrl_params_typ;
		parSw : stThicknessCtrl_paraSw;
		Outputs : stThicknessCtrl_ouputs_typ;
		Internal : stThicknessCtrl_Internal_typ;
		Alarms : stThicknessCtrl_Alarms_typ;
		AlSummary : stEFI_AlarmSummary;
	END_STRUCT;
END_TYPE
```

### Program Logical/ExtPack/_Media/ThicknessCtrl/ThicknessCtrl_v2/ThicknessCtrl (IEC)

#### ThicknessCtrl.st - Thickness detection & control
```iecst
PROGRAM _INIT

	RTInfo_0(enable :=TRUE );
	rPeriode:= UDINT_TO_REAL (RTInfo_0.cycle_time)/1000;  // Cycle time in microseconds

	//It is not controlled here rCycleFast to be here at this position, but if here is 0 is because the configuration is wrong
	gThicknessCtrl.Internal.rCycleSlow := rPeriode;
	gThicknessCtrl.Internal.rFastValues := gThicknessCtrl.Internal.rCycleSlow / gThicknessCtrl.Internal.rCycleFast;
	gThicknessCtrl.Internal.iFastValues := REAL_TO_UINT(gThicknessCtrl.Internal.rFastValues);

	// Moved here to assign internal arrays during initialization. Not needed aftewards in execution because just exists one instance of this program
	dataHeigh ACCESS ADR(gThicknessCtrl);

	MediaTrackingInsideL1 ACCESS ADR(dataHeigh.status.MediaPosition.L1.InsideMedia);
	MediaTrackingInsideL2 ACCESS ADR(dataHeigh.status.MediaPosition.L2.InsideMedia);

	//Assigning pointers here. Te position of the entering element is always the first one
	EnteringMediaL1 ACCESS ADR(MediaTrackingInsideL1[0]);
	EnteringMediaL2 ACCESS ADR(MediaTrackingInsideL2[0]);

	// iHeightArray initialization
	FOR iIndex := 0 TO iMAXHEIGHTARRAY DO
		iHeightArray[iIndex] := 1000; // 100.0 mm as initial value to avoid going to 0 height if the belt has not been moved
	END_FOR;

	EnergyTest.Energy.iPower[0,1] := EnergyTest.Energy.iPower[0,1];

	dataHeigh.Internal.pMediaTracking := ADR(xMediaTracking);
	dataHeigh.Internal.pDistanceWorkEmptyBelt := ADR(iDistanceWorkEmptyBelt);

END_PROGRAM

PROGRAM _CYCLIC

	// Assignation of """dataHeigh ACCESS ADR(gThicknessCtrl);""" is done in _INIT code

	//Limitation of the parameter
	CheckLimits;

	// Receive information of Media through OpcUa Method
	StackMethods;

	//Reset Alarms
	IF dataHeigh.Commands.xErrorRst THEN
		dataHeigh.Alarms := stAlarmsReseted;
		dataHeigh.AlSummary := stAlarmsSummaryReseted;
	END_IF

	//Thickness device is ready to detect media
	dataHeigh.status.DetectionSystem.xInPosition := (gDing.State.xDingInstalled OR gPhotoCells.status.xInPosition);

	// Adding the alarms to the mounted media consideration here, we gain 1 cycle in the machine fast to react
	xMountedMedia := gPhotoCells.status.xMountedMediaDetected OR gDing.State.xMountedMediaDetected OR
				gPhotoCells.Alarms.xMountedTile OR gPhotoCells.Alarms.xMountedTile OR gBasicDetectMedia.Alarms.xMountedMedia;

	// Update the value of the Height in the array if commanded
	IF dataHeigh.Commands.xAddSafetyMarginToHeight AND NOT xAddedSafetyMarginToHeight AND dataHeigh.status.MediaPosition.xMediaInside THEN
		iSafetyMarginToHeight := REAL_TO_UINT(dataHeigh.parameters.rSafetyMarginToHeight*100);
		FOR iIndexArray := 1 TO iTotalBlocksLengh DO
			//Apply heigh values to all the positions. Just if the value is lower
			iHeightArray[iIndexArray] := iHeightArray[iIndexArray] + iSafetyMarginToHeight;
		END_FOR
		xAddedSafetyMarginToHeight := TRUE;
	END_IF

	IF dataHeigh.Commands.UpdateAllMatrix OR dataHeigh.Commands.xAddSafetyMarginToHeight THEN
		ResetMaxHeigh;
		FOR iIndexArray := iTotalBlocksLengh TO 1 BY -1 DO
			//Apply heigh values to all the positions. Just if the value is lower
			iHeightArray[iIndexArray]:= MAX(iHeightArray[iIndexArray], iMediaHeight);
			AssignMaxHeighIndex;
		END_FOR
	END_IF

	IF (dataHeigh.parameters.Belt.rBeltSpeed >= rMinBeltSpeedToStart) THEN

		// Avoid multiple activation of xAddSafetyMarginToHeight if stopped
		xAddedSafetyMarginToHeight := FALSE;

		//Here we add the accumulated mm in the belt. Calculating the distance in ¿¿¿mm??? from speed (m/min x10) and the time in micros
		rAccumAdvBelt:= rAccumAdvBelt + dataHeigh.parameters.Belt.rBeltSpeed * rPeriode / 60;

		//Detect the quantity of positions the array must be moved
		iPositionsToRunArray := TRUNC(rAccumAdvBelt/MM_PERPOSITION_IN_ARRAY);

		//Just readjust if the advance has been more than a position
		IF iPositionsToRunArray >0 THEN

			//Recalculate the remaining Belt advance for the next execution
			rAccumAdvBelt := rAccumAdvBelt - iPositionsToRunArray * MM_PERPOSITION_IN_ARRAY;

			//Reduce the value in the distances vars
			SubstracDistances;

			// ------------------------------------------------------------------
			// RUN and REVIEW the arrays moving the values and filling the begining
			RunHeightArray;

			//Run over "Media" and "ValidMedia" matrixs if configured
			RunMediaArray;

			IF dataHeigh.parameters.Reject.xRejectTracking THEN
				RunRejectArray;
				ReviewRejectActivation;
			END_IF

			IF dataHeigh.parameters.Cure.xEnableTracking OR dataHeigh.parameters.Cure.xEnableMediaTracking THEN
				RunCureArray;
				ReviewCuringActivation;
			END_IF

			IF dataHeigh.parameters.Dry.xEnableMediaTracking THEN
				ReviewDryActivation;
			END_IF

			LoadDistancesBeltRunning;

			IF NOT dataHeigh.parameters.AutoMode.xJamRecovery THEN
				AlarmsCheckMedia;
			END_IF

		END_IF

		BoardsBelowBlockManagement;

	ELSE
		// RESETTING OUTPUTS IF BELT STOPPED
		dataHeigh.status.Belt.iBeltTurns := 0;
		// Reject outputs
		dataHeigh.Outputs.xHoldReject:=FALSE;
		xHoldReject:=FALSE;

		// Curing outputs
		dataHeigh.status.MediaPosition.L1.White.xMediaInLedPosition := FALSE;
		dataHeigh.status.MediaPosition.L1.Color.xMediaInLedPosition := FALSE;
		dataHeigh.status.MediaPosition.L1.Primer.xMediaInLedPosition := FALSE;
		dataHeigh.status.MediaPosition.L1.xDetectionSystemIncoherence := FALSE;
		dataHeigh.status.MediaPosition.L2.White.xMediaInLedPosition := FALSE;
		dataHeigh.status.MediaPosition.L2.Color.xMediaInLedPosition := FALSE;
		dataHeigh.status.MediaPosition.L2.Primer.xMediaInLedPosition := FALSE;
		dataHeigh.status.MediaPosition.L2.xDetectionSystemIncoherence := FALSE;

	END_IF

	// Resetting the BaordsFromStart when starting the belt
	IF EDGEPOS(dataHeigh.parameters.Belt.rBeltSpeed >= rMinBeltSpeedToStart) THEN
		dataHeigh.status.Detection.iBoardsFromStartL1 := 0;
		dataHeigh.status.Detection.iBoardsFromStartL2 := 0;
	END_IF

	LoadDistancesAlways;

	Alarms;

	AlarmSounds;

	AlarmsSummary;

	ReviewDryManual;

	//Reset counter if force
	IF dataHeigh.Commands.xResetMediaBelow THEN
		iBoardsBelowBlockL1:=0;
		iBoardsBelowBlockL2:=0;
		dataHeigh.status.Reject.iBoardsRejected := 0;
	END_IF
	IF EDGEPOS(dataHeigh.parameters.xBlockInProperPrintingPosition) THEN
		//dataHeigh.status.Reject.iBoardsRejected := 0;
		AddMediaTrackingEvents(diTotalCmBelt, END_REJECTING_ALL, ADR(TrackingEventsArray));
	END_IF
	IF EDGENEG(dataHeigh.parameters.xBlockInProperPrintingPosition) THEN
		AddMediaTrackingEvents(diTotalCmBelt, START_REJECTING_ALL, ADR(TrackingEventsArray));
	END_IF

	//TBD how reset will be activated
	tonResetRushProofCounterTimer.IN := dataHeigh.Commands.xErrorRst;
	tonResetRushProofCounterTimer.PT := T#5s;
	tonResetRushProofCounterTimer();
	xResetRejectRushProofCounter := tonResetRushProofCounterTimer.Q;
	IF xResetRejectRushProofCounter THEN
		iRushProofCounter:=0;
	END_IF

	// Empty belt state
	dataHeigh.status.Belt.xBeltEmpty:=iDistanceWorkEmptyBelt = 0;
	dataHeigh.status.MediaPosition.xMediaInside:=iDistanceMediaInside > 0;
	dataHeigh.status.MediaPosition.xTrackingEmpty := iDistanceTrackingEmpty = 0;
	dataHeigh.status.MediaPosition.xVirtualMediaInside:=iDistanceVirtualMediaInside > 0;
	dataHeigh.status.MediaPosition.xMediaToRejectInside := iDistanceMediaToRejectInside > 0;

	iReasonMediaBelow.0 := iDistanceMediaInside > 0;
	iReasonMediaBelow.1 := iDistanceVirtualMediaInside > 0;
	IF iReasonMediaBelow > 0 THEN
		dataHeigh.status.MediaPosition.xMediaBelowMachine:=TRUE;
	ELSIF NOT dataHeigh.status.MediaPosition.xMediaInside THEN
		dataHeigh.status.MediaPosition.xMediaBelowMachine:=FALSE;
	END_IF

	//If this value is higher than 0 is because still the belt has not been empty after a mounted alarm
	dataHeigh.status.MediaPosition.xMountedMediaInside 	:= iDistanceMountPieceOut>0;

	//To know when there is media at the end of printer's belt. Useful info for devices located afterwards (as Dryer)
	dataHeigh.status.MediaPosition.xMediaAtPrinterExit := xMediaTracking[dataHeigh.parameters.Belt.iDistanceEmptyBeltIni + 1] > 0;

	//Convert the internal value to the status value for beeing used in the printer
	LoadSectionsInformation;

	//Enabling PD signal to the carriage boards
	//Setting when PD signal positive edge and block is not at safe position or going back down printing position.
	dataHeigh.Outputs.xEnableMediaSignalToCb := dataHeigh.parameters.xBlockInProperPrintingPosition;

	//Media present in warp sensor position
	//Loading data
	dataHeigh.status.MediaPosition.xMediaInWarpSensorPosition := xFilteredAnalogSensorMedia OR xFilteredArraySensorMedia OR xFilteredBasicDetectionMedia;

	dataHeigh.status.xNewMediaStackEnabled := dataHeigh.parameters.Detection.xEnabledStack OR dataHeigh.parameters.Dry.xDryStack;
	dataHeigh.status.xMediaTrackingEnabled := dataHeigh.status.xNewMediaStackEnabled OR dataHeigh.parameters.Cure.xEnableMediaTracking OR dataHeigh.parameters.Dry.xEnableMediaTracking;

	// Define the MediaThickness margin to allow use it from outside
	IF NOT dataHeigh.status.xNewMediaStackEnabled THEN
		dataHeigh.status.Heigh.rMediaThicknessMargin := EnteringMediaContinuous.Media.rThickness + EnteringMediaContinuous.Media.rMargin;
		dataHeigh.status.Heigh.rMediaThickness 		 := EnteringMediaContinuous.Media.rThickness;
	ELSE
		rMediaThicknessMargin := 0;
		rMediaThickness := 0;
		IF MediaTracking_iTotalInsideL1 > 0 THEN // = ] := NewMediaStackL1[0];
			rMediaThicknessMargin := EnteringMediaL1.Media.rThickness + EnteringMediaL1.Media.rMargin;
			rMediaThickness := EnteringMediaL1.Media.rThickness;
		ELSE
			rMediaThicknessMargin := NewMediaStackL1[0].Media.rThickness + NewMediaStackL1[0].Media.rMargin;
			rMediaThickness := NewMediaStackL1[0].Media.rThickness;
		END_IF
		IF MediaTracking_iTotalInsideL2 > 0 THEN
			rMediaThicknessMargin := MAX(rMediaThicknessMargin, EnteringMediaL2.Media.rThickness + EnteringMediaL2.Media.rMargin);
			rMediaThickness := MAX(rMediaThickness, EnteringMediaL2.Media.rThickness + EnteringMediaL2.Media.rMargin);
		ELSE
			rMediaThicknessMargin := MAX(rMediaThicknessMargin, NewMediaStackL2[0].Media.rThickness + NewMediaStackL2[0].Media.rMargin);
			rMediaThickness := MAX(rMediaThickness, NewMediaStackL2[0].Media.rThickness + NewMediaStackL2[0].Media.rMargin);
		END_IF

		dataHeigh.status.Heigh.rMediaThicknessMargin := rMediaThicknessMargin;
		dataHeigh.status.Heigh.rMediaThickness := rMediaThickness;
	END_IF

	IF EDGEPOS(dataHeigh.status.MediaPosition.xMediaToRejectInside) THEN
		dataHeigh.status.Reject.iTimesInRejection := dataHeigh.status.Reject.iTimesInRejection + 1;
		dataHeigh.status.Reject.iTimesInRejectionToday := dataHeigh.status.Reject.iTimesInRejectionToday + 1;
	ELSIF EDGENEG(dataHeigh.status.MediaPosition.xMediaToRejectInside) THEN
		LogRejectingEnded;
	END_IF
	IF EDGEPOS(dataHeigh.parameters.AutoMode.xProduction) THEN // Changing to resetting when going into producion, to allow reading the value after stop
		dataHeigh.status.Reject.iTimesInRejection := 0;
	END_IF
	IF (tiTimeOfDay.hour = 0 AND tiTimeOfDay.hour = 0 AND tiTimeOfDay.minute = 0 AND tiTimeOfDay.second = 0) THEN
		dataHeigh.status.Reject.iTimesInRejectionToday := 0;
	END_IF

	// Getting time of the day
	GetTOD.enable := TRUE;
	GetTOD.pDTStructure := ADR(tiTimeOfDay);
	GetTOD();

	dataHeigh.Commands := CommandsReseted;
	xExitingMediaL1 := FALSE;
	xExitingMediaL2 := FALSE;

END_PROGRAM
```

#### CheckLimits.st
```iecst
ACTION CheckLimits:

	dataHeigh.status.Heigh.rMediaHeigh := UINT_TO_REAL(dataHeigh.status.Heigh.iMediaHeigh) / 100;
	iMediaHeight:= dataHeigh.status.Heigh.iMediaHeigh;

	iTotalSections := LIMIT(1, dataHeigh.parameters.iSections ,TOTAL_THICKNESS_SECTIONS);

	iTotalBlocksLengh := LIMIT(100, dataHeigh.parameters.iTotalBlocksLengh, iMAXHEIGHTARRAY);

	iRejectLengthAdjustment := LIMIT(100, dataHeigh.parameters.Belt.iDistanceEmptyBeltIni + dataHeigh.parameters.Reject.iRejectDistance, iMAXTRACKINGARRAY);
	iHoldRejectLengthAdjustment := LIMIT(100, dataHeigh.parameters.Belt.iDistanceEmptyBeltIni + dataHeigh.parameters.Reject.iHoldRejectDistance, iMAXTRACKINGARRAY);
	iMaxTrackingPosition := MAX(iRejectLengthAdjustment, iHoldRejectLengthAdjustment);
	FOR iIndexCheck:=1 TO MAX_LAST_CHECKMEDIA DO
		IF dataHeigh.parameters.CheckMedia[iIndexCheck].xActive THEN
			iMaxTrackingPosition := MAX(iMaxTrackingPosition, dataHeigh.parameters.CheckMedia[iIndexCheck].CheckPosition + dataHeigh.parameters.CheckMedia[iIndexCheck].CheckDelayPosition);
		END_IF
	END_FOR

	rMinBeltSpeedToStart := MAX(dataHeigh.parameters.Belt.rMinBeltSpeedToStart, 1.0);

	dataHeigh.Internal.rMarginSafePrintChecked := MAX(dataHeigh.parameters.rMarginSafePrint, 1.0); //The minimum Margin Safe print is 1mm

	iProductDetectSensorPosition := MIN(dataHeigh.parameters.Detection.ProductDetect.iSensorPosition, iMAXMEDIAPRESENTARRAY);
	iArraySensorPosition := MIN(dataHeigh.parameters.Detection.Array.iSensorPosition, iMAXMEDIAPRESENTARRAY);
	iAnalogSensorPosition := MIN(dataHeigh.parameters.Detection.Analog.iSensorPosition, iMAXMEDIAPRESENTARRAY);
	iDetectionMediaSensorPosition := MIN(dataHeigh.parameters.Detection.Basic.iSensorPosition, iMAXMEDIAPRESENTARRAY);
	iMediaFilter := MIN(dataHeigh.parameters.Detection.ProductDetect.iMediaFilter, 30);

	dataHeigh.parameters.Dry.rDryExtend := LIMIT(0,dataHeigh.parameters.Dry.rDryExtend, 100);

	//Limits for the array used with them
	iLastPosition := MAX(iTotalBlocksLengh, dataHeigh.parameters.Cure.White.iEndWindow, dataHeigh.parameters.Cure.Color.iEndWindow);
	iLastPosition := LIMIT(1, iLastPosition, iMAXTRACKINGARRAY);

END_ACTION
```
